; Data for Routine_1
DECL LDAT LCPDATP97={VEL 1.0,ACC 100,APO_DIST 5,APO_FAC 50.0,ORI_TYP #VAR,CIRC_TYP #BASE,JERK_FAC 50.0}
DECL FDAT FP97={TOOL_NO 2,BASE_NO 9,IPO_FRAME #BASE,POINT2[] " ",TQ_STATE FALSE}
DECL E6POS XP97={X 100.000,Y 0.000,Z -100.000,A 0.000,B 0.000,C 0.000}
DECL LDAT LCPDATP98={VEL 0.065,ACC 100,APO_DIST 5,APO_FAC 50.0,ORI_TYP #VAR,CIRC_TYP #BASE,JERK_FAC 50.0}
DECL FDAT FP98={TOOL_NO 2,BASE_NO 9,IPO_FRAME #BASE,POINT2[] " ",TQ_STATE FALSE}
DECL E6POS XP98={X 50.000,Y -2.120,Z -67.490,A 0.000,B 0.000,C -12.000}
DECL LDAT LCPDATP99={VEL 0.065,ACC 100,APO_DIST 5,APO_FAC 50.0,ORI_TYP #VAR,CIRC_TYP #BASE,JERK_FAC 50.0}
DECL FDAT FP99={TOOL_NO 2,BASE_NO 9,IPO_FRAME #BASE,POINT2[] " ",TQ_STATE FALSE}
DECL E6POS XP99={X 0.000,Y -2.120,Z -67.490,A 0.000,B 0.000,C -12.000}
DECL LDAT LCPDATP100={VEL 0.065,ACC 100,APO_DIST 5,APO_FAC 50.0,ORI_TYP #VAR,CIRC_TYP #BASE,JERK_FAC 50.0}
DECL FDAT FP100={TOOL_NO 2,BASE_NO 9,IPO_FRAME #BASE,POINT2[] " ",TQ_STATE FALSE}
DECL E6POS XP100={X -50.000,Y -2.120,Z -67.490,A 0.000,B 0.000,C -12.000}
DECL LDAT LCPDATP101={VEL 0.065,ACC 100,APO_DIST 5,APO_FAC 50.0,ORI_TYP #VAR,CIRC_TYP #BASE,JERK_FAC 50.0}
DECL FDAT FP101={TOOL_NO 2,BASE_NO 9,IPO_FRAME #BASE,POINT2[] " ",TQ_STATE FALSE}
DECL E6POS XP101={X -100.000,Y -2.120,Z -67.490,A 0.000,B 0.000,C -12.000}
DECL LDAT LCPDATP102={VEL 0.088,ACC 100,APO_DIST 5,APO_FAC 50.0,ORI_TYP #VAR,CIRC_TYP #BASE,JERK_FAC 50.0}
DECL FDAT FP102={TOOL_NO 2,BASE_NO 9,IPO_FRAME #BASE,POINT2[] " ",TQ_STATE FALSE}
DECL E6POS XP102={X -100.000,Y 15.760,Z -30.600,A 0.000,B 0.000,C -17.000}
DECL LDAT LCPDATP103={VEL 0.088,ACC 100,APO_DIST 5,APO_FAC 50.0,ORI_TYP #VAR,CIRC_TYP #BASE,JERK_FAC 50.0}
DECL FDAT FP103={TOOL_NO 2,BASE_NO 9,IPO_FRAME #BASE,POINT2[] " ",TQ_STATE FALSE}
DECL E6POS XP103={X -50.000,Y 15.760,Z -30.600,A 0.000,B 0.000,C -17.000}
DECL LDAT LCPDATP104={VEL 0.088,ACC 100,APO_DIST 5,APO_FAC 50.0,ORI_TYP #VAR,CIRC_TYP #BASE,JERK_FAC 50.0}
DECL FDAT FP104={TOOL_NO 2,BASE_NO 9,IPO_FRAME #BASE,POINT2[] " ",TQ_STATE FALSE}
DECL E6POS XP104={X -0.000,Y 15.760,Z -30.600,A 0.000,B 0.000,C -17.000}
DECL LDAT LCPDATP105={VEL 0.088,ACC 100,APO_DIST 5,APO_FAC 50.0,ORI_TYP #VAR,CIRC_TYP #BASE,JERK_FAC 50.0}
DECL FDAT FP105={TOOL_NO 2,BASE_NO 9,IPO_FRAME #BASE,POINT2[] " ",TQ_STATE FALSE}
DECL E6POS XP105={X 50.000,Y 15.760,Z -30.600,A 0.000,B 0.000,C -17.000}
DECL LDAT LCPDATP106={VEL 0.06,ACC 100,APO_DIST 5,APO_FAC 50.0,ORI_TYP #VAR,CIRC_TYP #BASE,JERK_FAC 50.0}
DECL FDAT FP106={TOOL_NO 2,BASE_NO 9,IPO_FRAME #BASE,POINT2[] " ",TQ_STATE FALSE}
DECL E6POS XP106={X 50.000,Y 13.210,Z -73.250,A 0.000,B 0.000,C -22.000}
DECL LDAT LCPDATP107={VEL 0.06,ACC 100,APO_DIST 5,APO_FAC 50.0,ORI_TYP #VAR,CIRC_TYP #BASE,JERK_FAC 50.0}
DECL FDAT FP107={TOOL_NO 2,BASE_NO 9,IPO_FRAME #BASE,POINT2[] " ",TQ_STATE FALSE}
DECL E6POS XP107={X -0.000,Y 13.210,Z -73.250,A 0.000,B 0.000,C -22.000}
DECL LDAT LCPDATP108={VEL 0.06,ACC 100,APO_DIST 5,APO_FAC 50.0,ORI_TYP #VAR,CIRC_TYP #BASE,JERK_FAC 50.0}
DECL FDAT FP108={TOOL_NO 2,BASE_NO 9,IPO_FRAME #BASE,POINT2[] " ",TQ_STATE FALSE}
DECL E6POS XP108={X -50.000,Y 13.210,Z -73.250,A 0.000,B 0.000,C -22.000}
DECL LDAT LCPDATP109={VEL 0.06,ACC 100,APO_DIST 5,APO_FAC 50.0,ORI_TYP #VAR,CIRC_TYP #BASE,JERK_FAC 50.0}
DECL FDAT FP109={TOOL_NO 2,BASE_NO 9,IPO_FRAME #BASE,POINT2[] " ",TQ_STATE FALSE}
DECL E6POS XP109={X -100.000,Y 13.210,Z -73.250,A 0.000,B 0.000,C -22.000}
DECL LDAT LCPDATP110={VEL 0.135,ACC 100,APO_DIST 5,APO_FAC 50.0,ORI_TYP #VAR,CIRC_TYP #BASE,JERK_FAC 50.0}
DECL FDAT FP110={TOOL_NO 2,BASE_NO 9,IPO_FRAME #BASE,POINT2[] " ",TQ_STATE FALSE}
DECL E6POS XP110={X -100.000,Y 40.110,Z -53.550,A 0.000,B 0.000,C -17.000}
DECL LDAT LCPDATP111={VEL 0.135,ACC 100,APO_DIST 5,APO_FAC 50.0,ORI_TYP #VAR,CIRC_TYP #BASE,JERK_FAC 50.0}
DECL FDAT FP111={TOOL_NO 2,BASE_NO 9,IPO_FRAME #BASE,POINT2[] " ",TQ_STATE FALSE}
DECL E6POS XP111={X -50.000,Y 40.110,Z -53.550,A 0.000,B 0.000,C -17.000}
DECL LDAT LCPDATP112={VEL 0.135,ACC 100,APO_DIST 5,APO_FAC 50.0,ORI_TYP #VAR,CIRC_TYP #BASE,JERK_FAC 50.0}
DECL FDAT FP112={TOOL_NO 2,BASE_NO 9,IPO_FRAME #BASE,POINT2[] " ",TQ_STATE FALSE}
DECL E6POS XP112={X -0.000,Y 40.110,Z -53.550,A 0.000,B 0.000,C -17.000}
DECL LDAT LCPDATP113={VEL 0.135,ACC 100,APO_DIST 5,APO_FAC 50.0,ORI_TYP #VAR,CIRC_TYP #BASE,JERK_FAC 50.0}
DECL FDAT FP113={TOOL_NO 2,BASE_NO 9,IPO_FRAME #BASE,POINT2[] " ",TQ_STATE FALSE}
DECL E6POS XP113={X 50.000,Y 40.110,Z -53.550,A 0.000,B 0.000,C -17.000}
DECL LDAT LCPDATP114={VEL 0.119,ACC 100,APO_DIST 5,APO_FAC 50.0,ORI_TYP #VAR,CIRC_TYP #BASE,JERK_FAC 50.0}
DECL FDAT FP114={TOOL_NO 2,BASE_NO 9,IPO_FRAME #BASE,POINT2[] " ",TQ_STATE FALSE}
DECL E6POS XP114={X 50.000,Y 24.230,Z -59.840,A 0.000,B 0.000,C -39.000}
DECL LDAT LCPDATP115={VEL 0.119,ACC 100,APO_DIST 5,APO_FAC 50.0,ORI_TYP #VAR,CIRC_TYP #BASE,JERK_FAC 50.0}
DECL FDAT FP115={TOOL_NO 2,BASE_NO 9,IPO_FRAME #BASE,POINT2[] " ",TQ_STATE FALSE}
DECL E6POS XP115={X -0.000,Y 24.230,Z -59.840,A 0.000,B 0.000,C -39.000}
DECL LDAT LCPDATP116={VEL 0.119,ACC 100,APO_DIST 5,APO_FAC 50.0,ORI_TYP #VAR,CIRC_TYP #BASE,JERK_FAC 50.0}
DECL FDAT FP116={TOOL_NO 2,BASE_NO 9,IPO_FRAME #BASE,POINT2[] " ",TQ_STATE FALSE}
DECL E6POS XP116={X -50.000,Y 24.230,Z -59.840,A 0.000,B 0.000,C -39.000}
DECL LDAT LCPDATP117={VEL 0.119,ACC 100,APO_DIST 5,APO_FAC 50.0,ORI_TYP #VAR,CIRC_TYP #BASE,JERK_FAC 50.0}
DECL FDAT FP117={TOOL_NO 2,BASE_NO 9,IPO_FRAME #BASE,POINT2[] " ",TQ_STATE FALSE}
DECL E6POS XP117={X -100.000,Y 24.230,Z -59.840,A 0.000,B 0.000,C -39.000}
DECL LDAT LCPDATP118={VEL 0.069,ACC 100,APO_DIST 5,APO_FAC 50.0,ORI_TYP #VAR,CIRC_TYP #BASE,JERK_FAC 50.0}
DECL FDAT FP118={TOOL_NO 2,BASE_NO 9,IPO_FRAME #BASE,POINT2[] " ",TQ_STATE FALSE}
DECL E6POS XP118={X -100.000,Y 48.790,Z -52.590,A 0.000,B 0.000,C -36.000}
DECL LDAT LCPDATP119={VEL 0.069,ACC 100,APO_DIST 5,APO_FAC 50.0,ORI_TYP #VAR,CIRC_TYP #BASE,JERK_FAC 50.0}
DECL FDAT FP119={TOOL_NO 2,BASE_NO 9,IPO_FRAME #BASE,POINT2[] " ",TQ_STATE FALSE}
DECL E6POS XP119={X -50.000,Y 48.790,Z -52.590,A 0.000,B 0.000,C -36.000}
DECL LDAT LCPDATP120={VEL 0.069,ACC 100,APO_DIST 5,APO_FAC 50.0,ORI_TYP #VAR,CIRC_TYP #BASE,JERK_FAC 50.0}
DECL FDAT FP120={TOOL_NO 2,BASE_NO 9,IPO_FRAME #BASE,POINT2[] " ",TQ_STATE FALSE}
DECL E6POS XP120={X -0.000,Y 48.790,Z -52.590,A 0.000,B 0.000,C -36.000}
DECL LDAT LCPDATP121={VEL 0.069,ACC 100,APO_DIST 5,APO_FAC 50.0,ORI_TYP #VAR,CIRC_TYP #BASE,JERK_FAC 50.0}
DECL FDAT FP121={TOOL_NO 2,BASE_NO 9,IPO_FRAME #BASE,POINT2[] " ",TQ_STATE FALSE}
DECL E6POS XP121={X 50.000,Y 48.790,Z -52.590,A 0.000,B 0.000,C -36.000}
DECL LDAT LCPDATP122={VEL 0.093,ACC 100,APO_DIST 5,APO_FAC 50.0,ORI_TYP #VAR,CIRC_TYP #BASE,JERK_FAC 50.0}
DECL FDAT FP122={TOOL_NO 2,BASE_NO 9,IPO_FRAME #BASE,POINT2[] " ",TQ_STATE FALSE}
DECL E6POS XP122={X 50.000,Y 91.140,Z -71.110,A 0.000,B 0.000,C -9.000}
DECL LDAT LCPDATP123={VEL 0.093,ACC 100,APO_DIST 5,APO_FAC 50.0,ORI_TYP #VAR,CIRC_TYP #BASE,JERK_FAC 50.0}
DECL FDAT FP123={TOOL_NO 2,BASE_NO 9,IPO_FRAME #BASE,POINT2[] " ",TQ_STATE FALSE}
DECL E6POS XP123={X -0.000,Y 91.140,Z -71.110,A 0.000,B 0.000,C -9.000}
DECL LDAT LCPDATP124={VEL 0.093,ACC 100,APO_DIST 5,APO_FAC 50.0,ORI_TYP #VAR,CIRC_TYP #BASE,JERK_FAC 50.0}
DECL FDAT FP124={TOOL_NO 2,BASE_NO 9,IPO_FRAME #BASE,POINT2[] " ",TQ_STATE FALSE}
DECL E6POS XP124={X -50.000,Y 91.140,Z -71.110,A 0.000,B 0.000,C -9.000}
DECL LDAT LCPDATP125={VEL 0.093,ACC 100,APO_DIST 5,APO_FAC 50.0,ORI_TYP #VAR,CIRC_TYP #BASE,JERK_FAC 50.0}
DECL FDAT FP125={TOOL_NO 2,BASE_NO 9,IPO_FRAME #BASE,POINT2[] " ",TQ_STATE FALSE}
DECL E6POS XP125={X -100.000,Y 91.140,Z -71.110,A 0.000,B 0.000,C -9.000}
DECL LDAT LCPDATP126={VEL 0.072,ACC 100,APO_DIST 5,APO_FAC 50.0,ORI_TYP #VAR,CIRC_TYP #BASE,JERK_FAC 50.0}
DECL FDAT FP126={TOOL_NO 2,BASE_NO 9,IPO_FRAME #BASE,POINT2[] " ",TQ_STATE FALSE}
DECL E6POS XP126={X -100.000,Y 100.110,Z -53.550,A 0.000,B 0.000,C -17.000}
DECL LDAT LCPDATP127={VEL 0.072,ACC 100,APO_DIST 5,APO_FAC 50.0,ORI_TYP #VAR,CIRC_TYP #BASE,JERK_FAC 50.0}
DECL FDAT FP127={TOOL_NO 2,BASE_NO 9,IPO_FRAME #BASE,POINT2[] " ",TQ_STATE FALSE}
DECL E6POS XP127={X -50.000,Y 100.110,Z -53.550,A 0.000,B 0.000,C -17.000}
DECL LDAT LCPDATP128={VEL 0.072,ACC 100,APO_DIST 5,APO_FAC 50.0,ORI_TYP #VAR,CIRC_TYP #BASE,JERK_FAC 50.0}
DECL FDAT FP128={TOOL_NO 2,BASE_NO 9,IPO_FRAME #BASE,POINT2[] " ",TQ_STATE FALSE}
DECL E6POS XP128={X -0.000,Y 100.110,Z -53.550,A 0.000,B 0.000,C -17.000}
DECL LDAT LCPDATP129={VEL 0.072,ACC 100,APO_DIST 5,APO_FAC 50.0,ORI_TYP #VAR,CIRC_TYP #BASE,JERK_FAC 50.0}
DECL FDAT FP129={TOOL_NO 2,BASE_NO 9,IPO_FRAME #BASE,POINT2[] " ",TQ_STATE FALSE}
DECL E6POS XP129={X 50.000,Y 100.110,Z -53.550,A 0.000,B 0.000,C -17.000}
DECL LDAT LCPDATP130={VEL 0.148,ACC 100,APO_DIST 5,APO_FAC 50.0,ORI_TYP #VAR,CIRC_TYP #BASE,JERK_FAC 50.0}
DECL FDAT FP130={TOOL_NO 2,BASE_NO 9,IPO_FRAME #BASE,POINT2[] " ",TQ_STATE FALSE}
DECL E6POS XP130={X 50.000,Y 97.570,Z -52.840,A 0.000,B 0.000,C -33.000}
DECL LDAT LCPDATP131={VEL 0.148,ACC 100,APO_DIST 5,APO_FAC 50.0,ORI_TYP #VAR,CIRC_TYP #BASE,JERK_FAC 50.0}
DECL FDAT FP131={TOOL_NO 2,BASE_NO 9,IPO_FRAME #BASE,POINT2[] " ",TQ_STATE FALSE}
DECL E6POS XP131={X -0.000,Y 97.570,Z -52.840,A 0.000,B 0.000,C -33.000}
DECL LDAT LCPDATP132={VEL 0.148,ACC 100,APO_DIST 5,APO_FAC 50.0,ORI_TYP #VAR,CIRC_TYP #BASE,JERK_FAC 50.0}
DECL FDAT FP132={TOOL_NO 2,BASE_NO 9,IPO_FRAME #BASE,POINT2[] " ",TQ_STATE FALSE}
DECL E6POS XP132={X -50.000,Y 97.570,Z -52.840,A 0.000,B 0.000,C -33.000}
DECL LDAT LCPDATP133={VEL 0.148,ACC 100,APO_DIST 5,APO_FAC 50.0,ORI_TYP #VAR,CIRC_TYP #BASE,JERK_FAC 50.0}
DECL FDAT FP133={TOOL_NO 2,BASE_NO 9,IPO_FRAME #BASE,POINT2[] " ",TQ_STATE FALSE}
DECL E6POS XP133={X -100.000,Y 97.570,Z -52.840,A 0.000,B 0.000,C -33.000}
DECL LDAT LCPDATP134={VEL 0.055,ACC 100,APO_DIST 5,APO_FAC 50.0,ORI_TYP #VAR,CIRC_TYP #BASE,JERK_FAC 50.0}
DECL FDAT FP134={TOOL_NO 2,BASE_NO 9,IPO_FRAME #BASE,POINT2[] " ",TQ_STATE FALSE}
DECL E6POS XP134={X -100.000,Y 134.600,Z -45.600,A 0.000,B 0.000,C -14.000}
DECL LDAT LCPDATP135={VEL 0.055,ACC 100,APO_DIST 5,APO_FAC 50.0,ORI_TYP #VAR,CIRC_TYP #BASE,JERK_FAC 50.0}
DECL FDAT FP135={TOOL_NO 2,BASE_NO 9,IPO_FRAME #BASE,POINT2[] " ",TQ_STATE FALSE}
DECL E6POS XP135={X -50.000,Y 134.600,Z -45.600,A 0.000,B 0.000,C -14.000}
DECL LDAT LCPDATP136={VEL 0.055,ACC 100,APO_DIST 5,APO_FAC 50.0,ORI_TYP #VAR,CIRC_TYP #BASE,JERK_FAC 50.0}
DECL FDAT FP136={TOOL_NO 2,BASE_NO 9,IPO_FRAME #BASE,POINT2[] " ",TQ_STATE FALSE}
DECL E6POS XP136={X -0.000,Y 134.600,Z -45.600,A 0.000,B 0.000,C -14.000}
DECL LDAT LCPDATP137={VEL 0.055,ACC 100,APO_DIST 5,APO_FAC 50.0,ORI_TYP #VAR,CIRC_TYP #BASE,JERK_FAC 50.0}
DECL FDAT FP137={TOOL_NO 2,BASE_NO 9,IPO_FRAME #BASE,POINT2[] " ",TQ_STATE FALSE}
DECL E6POS XP137={X 50.000,Y 134.600,Z -45.600,A 0.000,B 0.000,C -14.000}
DECL LDAT LCPDATP138={VEL 0.149,ACC 100,APO_DIST 5,APO_FAC 50.0,ORI_TYP #VAR,CIRC_TYP #BASE,JERK_FAC 50.0}
DECL FDAT FP138={TOOL_NO 2,BASE_NO 9,IPO_FRAME #BASE,POINT2[] " ",TQ_STATE FALSE}
DECL E6POS XP138={X 50.000,Y 142.850,Z -89.640,A 0.000,B 0.000,C -13.000}
DECL LDAT LCPDATP139={VEL 0.149,ACC 100,APO_DIST 5,APO_FAC 50.0,ORI_TYP #VAR,CIRC_TYP #BASE,JERK_FAC 50.0}
DECL FDAT FP139={TOOL_NO 2,BASE_NO 9,IPO_FRAME #BASE,POINT2[] " ",TQ_STATE FALSE}
DECL E6POS XP139={X -0.000,Y 142.850,Z -89.640,A 0.000,B 0.000,C -13.000}
DECL LDAT LCPDATP140={VEL 0.149,ACC 100,APO_DIST 5,APO_FAC 50.0,ORI_TYP #VAR,CIRC_TYP #BASE,JERK_FAC 50.0}
DECL FDAT FP140={TOOL_NO 2,BASE_NO 9,IPO_FRAME #BASE,POINT2[] " ",TQ_STATE FALSE}
DECL E6POS XP140={X -50.000,Y 142.850,Z -89.640,A 0.000,B 0.000,C -13.000}
DECL LDAT LCPDATP141={VEL 0.149,ACC 100,APO_DIST 5,APO_FAC 50.0,ORI_TYP #VAR,CIRC_TYP #BASE,JERK_FAC 50.0}
DECL FDAT FP141={TOOL_NO 2,BASE_NO 9,IPO_FRAME #BASE,POINT2[] " ",TQ_STATE FALSE}
DECL E6POS XP141={X -100.000,Y 142.850,Z -89.640,A 0.000,B 0.000,C -13.000}
DECL LDAT LCPDATP142={VEL 0.101,ACC 100,APO_DIST 5,APO_FAC 50.0,ORI_TYP #VAR,CIRC_TYP #BASE,JERK_FAC 50.0}
DECL FDAT FP142={TOOL_NO 2,BASE_NO 9,IPO_FRAME #BASE,POINT2[] " ",TQ_STATE FALSE}
DECL E6POS XP142={X -100.000,Y 141.950,Z -67.100,A 0.000,B 0.000,C -28.000}
DECL LDAT LCPDATP143={VEL 0.101,ACC 100,APO_DIST 5,APO_FAC 50.0,ORI_TYP #VAR,CIRC_TYP #BASE,JERK_FAC 50.0}
DECL FDAT FP143={TOOL_NO 2,BASE_NO 9,IPO_FRAME #BASE,POINT2[] " ",TQ_STATE FALSE}
DECL E6POS XP143={X -50.000,Y 141.950,Z -67.100,A 0.000,B 0.000,C -28.000}
DECL LDAT LCPDATP144={VEL 0.101,ACC 100,APO_DIST 5,APO_FAC 50.0,ORI_TYP #VAR,CIRC_TYP #BASE,JERK_FAC 50.0}
DECL FDAT FP144={TOOL_NO 2,BASE_NO 9,IPO_FRAME #BASE,POINT2[] " ",TQ_STATE FALSE}
DECL E6POS XP144={X -0.000,Y 141.950,Z -67.100,A 0.000,B 0.000,C -28.000}
DECL LDAT LCPDATP145={VEL 0.101,ACC 100,APO_DIST 5,APO_FAC 50.0,ORI_TYP #VAR,CIRC_TYP #BASE,JERK_FAC 50.0}
DECL FDAT FP145={TOOL_NO 2,BASE_NO 9,IPO_FRAME #BASE,POINT2[] " ",TQ_STATE FALSE}
DECL E6POS XP145={X 50.000,Y 141.950,Z -67.100,A 0.000,B 0.000,C -28.000}
DECL LDAT LCPDATP146={VEL 0.071,ACC 100,APO_DIST 5,APO_FAC 50.0,ORI_TYP #VAR,CIRC_TYP #BASE,JERK_FAC 50.0}
DECL FDAT FP146={TOOL_NO 2,BASE_NO 9,IPO_FRAME #BASE,POINT2[] " ",TQ_STATE FALSE}
DECL E6POS XP146={X 50.000,Y 189.020,Z -32.980,A 0.000,B 0.000,C -2.000}
DECL LDAT LCPDATP147={VEL 0.071,ACC 100,APO_DIST 5,APO_FAC 50.0,ORI_TYP #VAR,CIRC_TYP #BASE,JERK_FAC 50.0}
DECL FDAT FP147={TOOL_NO 2,BASE_NO 9,IPO_FRAME #BASE,POINT2[] " ",TQ_STATE FALSE}
DECL E6POS XP147={X -0.000,Y 189.020,Z -32.980,A 0.000,B 0.000,C -2.000}
DECL LDAT LCPDATP148={VEL 0.071,ACC 100,APO_DIST 5,APO_FAC 50.0,ORI_TYP #VAR,CIRC_TYP #BASE,JERK_FAC 50.0}
DECL FDAT FP148={TOOL_NO 2,BASE_NO 9,IPO_FRAME #BASE,POINT2[] " ",TQ_STATE FALSE}
DECL E6POS XP148={X -50.000,Y 189.020,Z -32.980,A 0.000,B 0.000,C -2.000}
DECL LDAT LCPDATP149={VEL 0.071,ACC 100,APO_DIST 5,APO_FAC 50.0,ORI_TYP #VAR,CIRC_TYP #BASE,JERK_FAC 50.0}
DECL FDAT FP149={TOOL_NO 2,BASE_NO 9,IPO_FRAME #BASE,POINT2[] " ",TQ_STATE FALSE}
DECL E6POS XP149={X -100.000,Y 189.020,Z -32.980,A 0.000,B 0.000,C -2.000}
DECL LDAT LCPDATP150={VEL 0.121,ACC 100,APO_DIST 5,APO_FAC 50.0,ORI_TYP #VAR,CIRC_TYP #BASE,JERK_FAC 50.0}
DECL FDAT FP150={TOOL_NO 2,BASE_NO 9,IPO_FRAME #BASE,POINT2[] " ",TQ_STATE FALSE}
DECL E6POS XP150={X -100.000,Y 199.670,Z -30.530,A 0.000,B 0.000,C -10.000}
DECL LDAT LCPDATP151={VEL 0.121,ACC 100,APO_DIST 5,APO_FAC 50.0,ORI_TYP #VAR,CIRC_TYP #BASE,JERK_FAC 50.0}
DECL FDAT FP151={TOOL_NO 2,BASE_NO 9,IPO_FRAME #BASE,POINT2[] " ",TQ_STATE FALSE}
DECL E6POS XP151={X -50.000,Y 199.670,Z -30.530,A 0.000,B 0.000,C -10.000}
DECL LDAT LCPDATP152={VEL 0.121,ACC 100,APO_DIST 5,APO_FAC 50.0,ORI_TYP #VAR,CIRC_TYP #BASE,JERK_FAC 50.0}
DECL FDAT FP152={TOOL_NO 2,BASE_NO 9,IPO_FRAME #BASE,POINT2[] " ",TQ_STATE FALSE}
DECL E6POS XP152={X -0.000,Y 199.670,Z -30.530,A 0.000,B 0.000,C -10.000}
DECL LDAT LCPDATP153={VEL 0.121,ACC 100,APO_DIST 5,APO_FAC 50.0,ORI_TYP #VAR,CIRC_TYP #BASE,JERK_FAC 50.0}
DECL FDAT FP153={TOOL_NO 2,BASE_NO 9,IPO_FRAME #BASE,POINT2[] " ",TQ_STATE FALSE}
DECL E6POS XP153={X 50.000,Y 199.670,Z -30.530,A 0.000,B 0.000,C -10.000}
DECL LDAT LCPDATP154={VEL 0.061,ACC 100,APO_DIST 5,APO_FAC 50.0,ORI_TYP #VAR,CIRC_TYP #BASE,JERK_FAC 50.0}
DECL FDAT FP154={TOOL_NO 2,BASE_NO 9,IPO_FRAME #BASE,POINT2[] " ",TQ_STATE FALSE}
DECL E6POS XP154={X 50.000,Y 202.790,Z -30.310,A 0.000,B 0.000,C -30.000}
DECL LDAT LCPDATP155={VEL 0.061,ACC 100,APO_DIST 5,APO_FAC 50.0,ORI_TYP #VAR,CIRC_TYP #BASE,JERK_FAC 50.0}
DECL FDAT FP155={TOOL_NO 2,BASE_NO 9,IPO_FRAME #BASE,POINT2[] " ",TQ_STATE FALSE}
DECL E6POS XP155={X -0.000,Y 202.790,Z -30.310,A 0.000,B 0.000,C -30.000}
DECL LDAT LCPDATP156={VEL 0.061,ACC 100,APO_DIST 5,APO_FAC 50.0,ORI_TYP #VAR,CIRC_TYP #BASE,JERK_FAC 50.0}
DECL FDAT FP156={TOOL_NO 2,BASE_NO 9,IPO_FRAME #BASE,POINT2[] " ",TQ_STATE FALSE}
DECL E6POS XP156={X -50.000,Y 202.790,Z -30.310,A 0.000,B 0.000,C -30.000}
DECL LDAT LCPDATP157={VEL 0.061,ACC 100,APO_DIST 5,APO_FAC 50.0,ORI_TYP #VAR,CIRC_TYP #BASE,JERK_FAC 50.0}
DECL FDAT FP157={TOOL_NO 2,BASE_NO 9,IPO_FRAME #BASE,POINT2[] " ",TQ_STATE FALSE}
DECL E6POS XP157={X -100.000,Y 202.790,Z -30.310,A 0.000,B 0.000,C -30.000}
DECL LDAT LCPDATP158={VEL 0.5,ACC 100,APO_DIST 5,APO_FAC 50.0,ORI_TYP #VAR,CIRC_TYP #BASE,JERK_FAC 50.0}
DECL FDAT FP158={TOOL_NO 2,BASE_NO 9,IPO_FRAME #BASE,POINT2[] " ",TQ_STATE FALSE}
DECL E6POS XP158={X -150.000,Y 220.290,Z -50.000,A 0.000,B 0.000,C 0.000}
DECL LDAT LCPDATP159={VEL 1.0,ACC 100,APO_DIST 5,APO_FAC 50.0,ORI_TYP #VAR,CIRC_TYP #BASE,JERK_FAC 50.0}
DECL FDAT FP159={TOOL_NO 2,BASE_NO 9,IPO_FRAME #BASE,POINT2[] " ",TQ_STATE FALSE}
DECL E6POS XP159={X -150.000,Y 260.000,Z -20.000,A 0.000,B 0.000,C 0.000}
DECL LDAT LCPDATP160={VEL 1.0,ACC 100,APO_DIST 5,APO_FAC 50.0,ORI_TYP #VAR,CIRC_TYP #BASE,JERK_FAC 50.0}
DECL FDAT FP160={TOOL_NO 2,BASE_NO 9,IPO_FRAME #BASE,POINT2[] " ",TQ_STATE FALSE}
DECL E6POS XP160={X 100.000,Y 260.000,Z -20.000,A 0.000,B 0.000,C 0.000}
;ENDDAT for Routine_1


; Data for Routine_2
DECL LDAT LCPDATP161={VEL 1.0,ACC 100,APO_DIST 5,APO_FAC 50.0,ORI_TYP #VAR,CIRC_TYP #BASE,JERK_FAC 50.0}
DECL FDAT FP161={TOOL_NO 2,BASE_NO 8,IPO_FRAME #BASE,POINT2[] " ",TQ_STATE FALSE}
DECL E6POS XP161={X 100.000,Y 0.000,Z -100.000,A 0.000,B 0.000,C 0.000}
DECL LDAT LCPDATP162={VEL 0.123,ACC 100,APO_DIST 5,APO_FAC 50.0,ORI_TYP #VAR,CIRC_TYP #BASE,JERK_FAC 50.0}
DECL FDAT FP162={TOOL_NO 2,BASE_NO 8,IPO_FRAME #BASE,POINT2[] " ",TQ_STATE FALSE}
DECL E6POS XP162={X 50.000,Y -12.510,Z -68.600,A 0.000,B 0.000,C -20.000}
DECL LDAT LCPDATP163={VEL 0.123,ACC 100,APO_DIST 5,APO_FAC 50.0,ORI_TYP #VAR,CIRC_TYP #BASE,JERK_FAC 50.0}
DECL FDAT FP163={TOOL_NO 2,BASE_NO 8,IPO_FRAME #BASE,POINT2[] " ",TQ_STATE FALSE}
DECL E6POS XP163={X 0.000,Y -12.510,Z -68.600,A 0.000,B 0.000,C -20.000}
DECL LDAT LCPDATP164={VEL 0.123,ACC 100,APO_DIST 5,APO_FAC 50.0,ORI_TYP #VAR,CIRC_TYP #BASE,JERK_FAC 50.0}
DECL FDAT FP164={TOOL_NO 2,BASE_NO 8,IPO_FRAME #BASE,POINT2[] " ",TQ_STATE FALSE}
DECL E6POS XP164={X -50.000,Y -12.510,Z -68.600,A 0.000,B 0.000,C -20.000}
DECL LDAT LCPDATP165={VEL 0.123,ACC 100,APO_DIST 5,APO_FAC 50.0,ORI_TYP #VAR,CIRC_TYP #BASE,JERK_FAC 50.0}
DECL FDAT FP165={TOOL_NO 2,BASE_NO 8,IPO_FRAME #BASE,POINT2[] " ",TQ_STATE FALSE}
DECL E6POS XP165={X -100.000,Y -12.510,Z -68.600,A 0.000,B 0.000,C -20.000}
DECL LDAT LCPDATP166={VEL 0.128,ACC 100,APO_DIST 5,APO_FAC 50.0,ORI_TYP #VAR,CIRC_TYP #BASE,JERK_FAC 50.0}
DECL FDAT FP166={TOOL_NO 2,BASE_NO 8,IPO_FRAME #BASE,POINT2[] " ",TQ_STATE FALSE}
DECL E6POS XP166={X -100.000,Y -8.150,Z -77.940,A 0.000,B 0.000,C -25.000}
DECL LDAT LCPDATP167={VEL 0.128,ACC 100,APO_DIST 5,APO_FAC 50.0,ORI_TYP #VAR,CIRC_TYP #BASE,JERK_FAC 50.0}
DECL FDAT FP167={TOOL_NO 2,BASE_NO 8,IPO_FRAME #BASE,POINT2[] " ",TQ_STATE FALSE}
DECL E6POS XP167={X -50.000,Y -8.150,Z -77.940,A 0.000,B 0.000,C -25.000}
DECL LDAT LCPDATP168={VEL 0.128,ACC 100,APO_DIST 5,APO_FAC 50.0,ORI_TYP #VAR,CIRC_TYP #BASE,JERK_FAC 50.0}
DECL FDAT FP168={TOOL_NO 2,BASE_NO 8,IPO_FRAME #BASE,POINT2[] " ",TQ_STATE FALSE}
DECL E6POS XP168={X 0.000,Y -8.150,Z -77.940,A 0.000,B 0.000,C -25.000}
DECL LDAT LCPDATP169={VEL 0.128,ACC 100,APO_DIST 5,APO_FAC 50.0,ORI_TYP #VAR,CIRC_TYP #BASE,JERK_FAC 50.0}
DECL FDAT FP169={TOOL_NO 2,BASE_NO 8,IPO_FRAME #BASE,POINT2[] " ",TQ_STATE FALSE}
DECL E6POS XP169={X 50.000,Y -8.150,Z -77.940,A 0.000,B 0.000,C -25.000}
DECL LDAT LCPDATP170={VEL 0.103,ACC 100,APO_DIST 5,APO_FAC 50.0,ORI_TYP #VAR,CIRC_TYP #BASE,JERK_FAC 50.0}
DECL FDAT FP170={TOOL_NO 2,BASE_NO 8,IPO_FRAME #BASE,POINT2[] " ",TQ_STATE FALSE}
DECL E6POS XP170={X 50.000,Y 41.710,Z -60.000,A 0.000,B 0.000,C 0.000}
DECL LDAT LCPDATP171={VEL 0.103,ACC 100,APO_DIST 5,APO_FAC 50.0,ORI_TYP #VAR,CIRC_TYP #BASE,JERK_FAC 50.0}
DECL FDAT FP171={TOOL_NO 2,BASE_NO 8,IPO_FRAME #BASE,POINT2[] " ",TQ_STATE FALSE}
DECL E6POS XP171={X -0.000,Y 41.710,Z -60.000,A 0.000,B 0.000,C 0.000}
DECL LDAT LCPDATP172={VEL 0.103,ACC 100,APO_DIST 5,APO_FAC 50.0,ORI_TYP #VAR,CIRC_TYP #BASE,JERK_FAC 50.0}
DECL FDAT FP172={TOOL_NO 2,BASE_NO 8,IPO_FRAME #BASE,POINT2[] " ",TQ_STATE FALSE}
DECL E6POS XP172={X -50.000,Y 41.710,Z -60.000,A 0.000,B 0.000,C 0.000}
DECL LDAT LCPDATP173={VEL 0.103,ACC 100,APO_DIST 5,APO_FAC 50.0,ORI_TYP #VAR,CIRC_TYP #BASE,JERK_FAC 50.0}
DECL FDAT FP173={TOOL_NO 2,BASE_NO 8,IPO_FRAME #BASE,POINT2[] " ",TQ_STATE FALSE}
DECL E6POS XP173={X -100.000,Y 41.710,Z -60.000,A 0.000,B 0.000,C 0.000}
DECL LDAT LCPDATP174={VEL 0.108,ACC 100,APO_DIST 5,APO_FAC 50.0,ORI_TYP #VAR,CIRC_TYP #BASE,JERK_FAC 50.0}
DECL FDAT FP174={TOOL_NO 2,BASE_NO 8,IPO_FRAME #BASE,POINT2[] " ",TQ_STATE FALSE}
DECL E6POS XP174={X -100.000,Y 43.810,Z -45.400,A 0.000,B 0.000,C -15.000}
DECL LDAT LCPDATP175={VEL 0.108,ACC 100,APO_DIST 5,APO_FAC 50.0,ORI_TYP #VAR,CIRC_TYP #BASE,JERK_FAC 50.0}
DECL FDAT FP175={TOOL_NO 2,BASE_NO 8,IPO_FRAME #BASE,POINT2[] " ",TQ_STATE FALSE}
DECL E6POS XP175={X -50.000,Y 43.810,Z -45.400,A 0.000,B 0.000,C -15.000}
DECL LDAT LCPDATP176={VEL 0.108,ACC 100,APO_DIST 5,APO_FAC 50.0,ORI_TYP #VAR,CIRC_TYP #BASE,JERK_FAC 50.0}
DECL FDAT FP176={TOOL_NO 2,BASE_NO 8,IPO_FRAME #BASE,POINT2[] " ",TQ_STATE FALSE}
DECL E6POS XP176={X -0.000,Y 43.810,Z -45.400,A 0.000,B 0.000,C -15.000}
DECL LDAT LCPDATP177={VEL 0.108,ACC 100,APO_DIST 5,APO_FAC 50.0,ORI_TYP #VAR,CIRC_TYP #BASE,JERK_FAC 50.0}
DECL FDAT FP177={TOOL_NO 2,BASE_NO 8,IPO_FRAME #BASE,POINT2[] " ",TQ_STATE FALSE}
DECL E6POS XP177={X 50.000,Y 43.810,Z -45.400,A 0.000,B 0.000,C -15.000}
DECL LDAT LCPDATP178={VEL 0.095,ACC 100,APO_DIST 5,APO_FAC 50.0,ORI_TYP #VAR,CIRC_TYP #BASE,JERK_FAC 50.0}
DECL FDAT FP178={TOOL_NO 2,BASE_NO 8,IPO_FRAME #BASE,POINT2[] " ",TQ_STATE FALSE}
DECL E6POS XP178={X 50.000,Y 50.270,Z -49.710,A 0.000,B 0.000,C -23.000}
DECL LDAT LCPDATP179={VEL 0.095,ACC 100,APO_DIST 5,APO_FAC 50.0,ORI_TYP #VAR,CIRC_TYP #BASE,JERK_FAC 50.0}
DECL FDAT FP179={TOOL_NO 2,BASE_NO 8,IPO_FRAME #BASE,POINT2[] " ",TQ_STATE FALSE}
DECL E6POS XP179={X -0.000,Y 50.270,Z -49.710,A 0.000,B 0.000,C -23.000}
DECL LDAT LCPDATP180={VEL 0.095,ACC 100,APO_DIST 5,APO_FAC 50.0,ORI_TYP #VAR,CIRC_TYP #BASE,JERK_FAC 50.0}
DECL FDAT FP180={TOOL_NO 2,BASE_NO 8,IPO_FRAME #BASE,POINT2[] " ",TQ_STATE FALSE}
DECL E6POS XP180={X -50.000,Y 50.270,Z -49.710,A 0.000,B 0.000,C -23.000}
DECL LDAT LCPDATP181={VEL 0.095,ACC 100,APO_DIST 5,APO_FAC 50.0,ORI_TYP #VAR,CIRC_TYP #BASE,JERK_FAC 50.0}
DECL FDAT FP181={TOOL_NO 2,BASE_NO 8,IPO_FRAME #BASE,POINT2[] " ",TQ_STATE FALSE}
DECL E6POS XP181={X -100.000,Y 50.270,Z -49.710,A 0.000,B 0.000,C -23.000}
DECL LDAT LCPDATP182={VEL 0.142,ACC 100,APO_DIST 5,APO_FAC 50.0,ORI_TYP #VAR,CIRC_TYP #BASE,JERK_FAC 50.0}
DECL FDAT FP182={TOOL_NO 2,BASE_NO 8,IPO_FRAME #BASE,POINT2[] " ",TQ_STATE FALSE}
DECL E6POS XP182={X -100.000,Y 77.240,Z -35.080,A 0.000,B 0.000,C -13.000}
DECL LDAT LCPDATP183={VEL 0.142,ACC 100,APO_DIST 5,APO_FAC 50.0,ORI_TYP #VAR,CIRC_TYP #BASE,JERK_FAC 50.0}
DECL FDAT FP183={TOOL_NO 2,BASE_NO 8,IPO_FRAME #BASE,POINT2[] " ",TQ_STATE FALSE}
DECL E6POS XP183={X -50.000,Y 77.240,Z -35.080,A 0.000,B 0.000,C -13.000}
DECL LDAT LCPDATP184={VEL 0.142,ACC 100,APO_DIST 5,APO_FAC 50.0,ORI_TYP #VAR,CIRC_TYP #BASE,JERK_FAC 50.0}
DECL FDAT FP184={TOOL_NO 2,BASE_NO 8,IPO_FRAME #BASE,POINT2[] " ",TQ_STATE FALSE}
DECL E6POS XP184={X -0.000,Y 77.240,Z -35.080,A 0.000,B 0.000,C -13.000}
DECL LDAT LCPDATP185={VEL 0.142,ACC 100,APO_DIST 5,APO_FAC 50.0,ORI_TYP #VAR,CIRC_TYP #BASE,JERK_FAC 50.0}
DECL FDAT FP185={TOOL_NO 2,BASE_NO 8,IPO_FRAME #BASE,POINT2[] " ",TQ_STATE FALSE}
DECL E6POS XP185={X 50.000,Y 77.240,Z -35.080,A 0.000,B 0.000,C -13.000}
DECL LDAT LCPDATP186={VEL 0.142,ACC 100,APO_DIST 5,APO_FAC 50.0,ORI_TYP #VAR,CIRC_TYP #BASE,JERK_FAC 50.0}
DECL FDAT FP186={TOOL_NO 2,BASE_NO 8,IPO_FRAME #BASE,POINT2[] " ",TQ_STATE FALSE}
DECL E6POS XP186={X 50.000,Y 94.780,Z -73.590,A 0.000,B 0.000,C -6.000}
DECL LDAT LCPDATP187={VEL 0.142,ACC 100,APO_DIST 5,APO_FAC 50.0,ORI_TYP #VAR,CIRC_TYP #BASE,JERK_FAC 50.0}
DECL FDAT FP187={TOOL_NO 2,BASE_NO 8,IPO_FRAME #BASE,POINT2[] " ",TQ_STATE FALSE}
DECL E6POS XP187={X -0.000,Y 94.780,Z -73.590,A 0.000,B 0.000,C -6.000}
DECL LDAT LCPDATP188={VEL 0.142,ACC 100,APO_DIST 5,APO_FAC 50.0,ORI_TYP #VAR,CIRC_TYP #BASE,JERK_FAC 50.0}
DECL FDAT FP188={TOOL_NO 2,BASE_NO 8,IPO_FRAME #BASE,POINT2[] " ",TQ_STATE FALSE}
DECL E6POS XP188={X -50.000,Y 94.780,Z -73.590,A 0.000,B 0.000,C -6.000}
DECL LDAT LCPDATP189={VEL 0.142,ACC 100,APO_DIST 5,APO_FAC 50.0,ORI_TYP #VAR,CIRC_TYP #BASE,JERK_FAC 50.0}
DECL FDAT FP189={TOOL_NO 2,BASE_NO 8,IPO_FRAME #BASE,POINT2[] " ",TQ_STATE FALSE}
DECL E6POS XP189={X -100.000,Y 94.780,Z -73.590,A 0.000,B 0.000,C -6.000}
DECL LDAT LCPDATP190={VEL 0.064,ACC 100,APO_DIST 5,APO_FAC 50.0,ORI_TYP #VAR,CIRC_TYP #BASE,JERK_FAC 50.0}
DECL FDAT FP190={TOOL_NO 2,BASE_NO 8,IPO_FRAME #BASE,POINT2[] " ",TQ_STATE FALSE}
DECL E6POS XP190={X -100.000,Y 84.800,Z -40.190,A 0.000,B 0.000,C -38.000}
DECL LDAT LCPDATP191={VEL 0.064,ACC 100,APO_DIST 5,APO_FAC 50.0,ORI_TYP #VAR,CIRC_TYP #BASE,JERK_FAC 50.0}
DECL FDAT FP191={TOOL_NO 2,BASE_NO 8,IPO_FRAME #BASE,POINT2[] " ",TQ_STATE FALSE}
DECL E6POS XP191={X -50.000,Y 84.800,Z -40.190,A 0.000,B 0.000,C -38.000}
DECL LDAT LCPDATP192={VEL 0.064,ACC 100,APO_DIST 5,APO_FAC 50.0,ORI_TYP #VAR,CIRC_TYP #BASE,JERK_FAC 50.0}
DECL FDAT FP192={TOOL_NO 2,BASE_NO 8,IPO_FRAME #BASE,POINT2[] " ",TQ_STATE FALSE}
DECL E6POS XP192={X -0.000,Y 84.800,Z -40.190,A 0.000,B 0.000,C -38.000}
DECL LDAT LCPDATP193={VEL 0.064,ACC 100,APO_DIST 5,APO_FAC 50.0,ORI_TYP #VAR,CIRC_TYP #BASE,JERK_FAC 50.0}
DECL FDAT FP193={TOOL_NO 2,BASE_NO 8,IPO_FRAME #BASE,POINT2[] " ",TQ_STATE FALSE}
DECL E6POS XP193={X 50.000,Y 84.800,Z -40.190,A 0.000,B 0.000,C -38.000}
DECL LDAT LCPDATP194={VEL 0.055,ACC 100,APO_DIST 5,APO_FAC 50.0,ORI_TYP #VAR,CIRC_TYP #BASE,JERK_FAC 50.0}
DECL FDAT FP194={TOOL_NO 2,BASE_NO 8,IPO_FRAME #BASE,POINT2[] " ",TQ_STATE FALSE}
DECL E6POS XP194={X 50.000,Y 76.790,Z -69.940,A 0.000,B 0.000,C -39.000}
DECL LDAT LCPDATP195={VEL 0.055,ACC 100,APO_DIST 5,APO_FAC 50.0,ORI_TYP #VAR,CIRC_TYP #BASE,JERK_FAC 50.0}
DECL FDAT FP195={TOOL_NO 2,BASE_NO 8,IPO_FRAME #BASE,POINT2[] " ",TQ_STATE FALSE}
DECL E6POS XP195={X -0.000,Y 76.790,Z -69.940,A 0.000,B 0.000,C -39.000}
DECL LDAT LCPDATP196={VEL 0.055,ACC 100,APO_DIST 5,APO_FAC 50.0,ORI_TYP #VAR,CIRC_TYP #BASE,JERK_FAC 50.0}
DECL FDAT FP196={TOOL_NO 2,BASE_NO 8,IPO_FRAME #BASE,POINT2[] " ",TQ_STATE FALSE}
DECL E6POS XP196={X -50.000,Y 76.790,Z -69.940,A 0.000,B 0.000,C -39.000}
DECL LDAT LCPDATP197={VEL 0.055,ACC 100,APO_DIST 5,APO_FAC 50.0,ORI_TYP #VAR,CIRC_TYP #BASE,JERK_FAC 50.0}
DECL FDAT FP197={TOOL_NO 2,BASE_NO 8,IPO_FRAME #BASE,POINT2[] " ",TQ_STATE FALSE}
DECL E6POS XP197={X -100.000,Y 76.790,Z -69.940,A 0.000,B 0.000,C -39.000}
DECL LDAT LCPDATP198={VEL 0.12,ACC 100,APO_DIST 5,APO_FAC 50.0,ORI_TYP #VAR,CIRC_TYP #BASE,JERK_FAC 50.0}
DECL FDAT FP198={TOOL_NO 2,BASE_NO 8,IPO_FRAME #BASE,POINT2[] " ",TQ_STATE FALSE}
DECL E6POS XP198={X -100.000,Y 132.190,Z -81.480,A 0.000,B 0.000,C -11.000}
DECL LDAT LCPDATP199={VEL 0.12,ACC 100,APO_DIST 5,APO_FAC 50.0,ORI_TYP #VAR,CIRC_TYP #BASE,JERK_FAC 50.0}
DECL FDAT FP199={TOOL_NO 2,BASE_NO 8,IPO_FRAME #BASE,POINT2[] " ",TQ_STATE FALSE}
DECL E6POS XP199={X -50.000,Y 132.190,Z -81.480,A 0.000,B 0.000,C -11.000}
DECL LDAT LCPDATP200={VEL 0.12,ACC 100,APO_DIST 5,APO_FAC 50.0,ORI_TYP #VAR,CIRC_TYP #BASE,JERK_FAC 50.0}
DECL FDAT FP200={TOOL_NO 2,BASE_NO 8,IPO_FRAME #BASE,POINT2[] " ",TQ_STATE FALSE}
DECL E6POS XP200={X -0.000,Y 132.190,Z -81.480,A 0.000,B 0.000,C -11.000}
DECL LDAT LCPDATP201={VEL 0.12,ACC 100,APO_DIST 5,APO_FAC 50.0,ORI_TYP #VAR,CIRC_TYP #BASE,JERK_FAC 50.0}
DECL FDAT FP201={TOOL_NO 2,BASE_NO 8,IPO_FRAME #BASE,POINT2[] " ",TQ_STATE FALSE}
DECL E6POS XP201={X 50.000,Y 132.190,Z -81.480,A 0.000,B 0.000,C -11.000}
DECL LDAT LCPDATP202={VEL 0.081,ACC 100,APO_DIST 5,APO_FAC 50.0,ORI_TYP #VAR,CIRC_TYP #BASE,JERK_FAC 50.0}
DECL FDAT FP202={TOOL_NO 2,BASE_NO 8,IPO_FRAME #BASE,POINT2[] " ",TQ_STATE FALSE}
DECL E6POS XP202={X 50.000,Y 124.070,Z -69.970,A 0.000,B 0.000,C -29.000}
DECL LDAT LCPDATP203={VEL 0.081,ACC 100,APO_DIST 5,APO_FAC 50.0,ORI_TYP #VAR,CIRC_TYP #BASE,JERK_FAC 50.0}
DECL FDAT FP203={TOOL_NO 2,BASE_NO 8,IPO_FRAME #BASE,POINT2[] " ",TQ_STATE FALSE}
DECL E6POS XP203={X -0.000,Y 124.070,Z -69.970,A 0.000,B 0.000,C -29.000}
DECL LDAT LCPDATP204={VEL 0.081,ACC 100,APO_DIST 5,APO_FAC 50.0,ORI_TYP #VAR,CIRC_TYP #BASE,JERK_FAC 50.0}
DECL FDAT FP204={TOOL_NO 2,BASE_NO 8,IPO_FRAME #BASE,POINT2[] " ",TQ_STATE FALSE}
DECL E6POS XP204={X -50.000,Y 124.070,Z -69.970,A 0.000,B 0.000,C -29.000}
DECL LDAT LCPDATP205={VEL 0.081,ACC 100,APO_DIST 5,APO_FAC 50.0,ORI_TYP #VAR,CIRC_TYP #BASE,JERK_FAC 50.0}
DECL FDAT FP205={TOOL_NO 2,BASE_NO 8,IPO_FRAME #BASE,POINT2[] " ",TQ_STATE FALSE}
DECL E6POS XP205={X -100.000,Y 124.070,Z -69.970,A 0.000,B 0.000,C -29.000}
DECL LDAT LCPDATP206={VEL 0.147,ACC 100,APO_DIST 5,APO_FAC 50.0,ORI_TYP #VAR,CIRC_TYP #BASE,JERK_FAC 50.0}
DECL FDAT FP206={TOOL_NO 2,BASE_NO 8,IPO_FRAME #BASE,POINT2[] " ",TQ_STATE FALSE}
DECL E6POS XP206={X -100.000,Y 170.770,Z -52.710,A 0.000,B 0.000,C -6.000}
DECL LDAT LCPDATP207={VEL 0.147,ACC 100,APO_DIST 5,APO_FAC 50.0,ORI_TYP #VAR,CIRC_TYP #BASE,JERK_FAC 50.0}
DECL FDAT FP207={TOOL_NO 2,BASE_NO 8,IPO_FRAME #BASE,POINT2[] " ",TQ_STATE FALSE}
DECL E6POS XP207={X -50.000,Y 170.770,Z -52.710,A 0.000,B 0.000,C -6.000}
DECL LDAT LCPDATP208={VEL 0.147,ACC 100,APO_DIST 5,APO_FAC 50.0,ORI_TYP #VAR,CIRC_TYP #BASE,JERK_FAC 50.0}
DECL FDAT FP208={TOOL_NO 2,BASE_NO 8,IPO_FRAME #BASE,POINT2[] " ",TQ_STATE FALSE}
DECL E6POS XP208={X -0.000,Y 170.770,Z -52.710,A 0.000,B 0.000,C -6.000}
DECL LDAT LCPDATP209={VEL 0.147,ACC 100,APO_DIST 5,APO_FAC 50.0,ORI_TYP #VAR,CIRC_TYP #BASE,JERK_FAC 50.0}
DECL FDAT FP209={TOOL_NO 2,BASE_NO 8,IPO_FRAME #BASE,POINT2[] " ",TQ_STATE FALSE}
DECL E6POS XP209={X 50.000,Y 170.770,Z -52.710,A 0.000,B 0.000,C -6.000}
DECL LDAT LCPDATP210={VEL 0.076,ACC 100,APO_DIST 5,APO_FAC 50.0,ORI_TYP #VAR,CIRC_TYP #BASE,JERK_FAC 50.0}
DECL FDAT FP210={TOOL_NO 2,BASE_NO 8,IPO_FRAME #BASE,POINT2[] " ",TQ_STATE FALSE}
DECL E6POS XP210={X 50.000,Y 145.240,Z -80.570,A 0.000,B 0.000,C -31.000}
DECL LDAT LCPDATP211={VEL 0.076,ACC 100,APO_DIST 5,APO_FAC 50.0,ORI_TYP #VAR,CIRC_TYP #BASE,JERK_FAC 50.0}
DECL FDAT FP211={TOOL_NO 2,BASE_NO 8,IPO_FRAME #BASE,POINT2[] " ",TQ_STATE FALSE}
DECL E6POS XP211={X -0.000,Y 145.240,Z -80.570,A 0.000,B 0.000,C -31.000}
DECL LDAT LCPDATP212={VEL 0.076,ACC 100,APO_DIST 5,APO_FAC 50.0,ORI_TYP #VAR,CIRC_TYP #BASE,JERK_FAC 50.0}
DECL FDAT FP212={TOOL_NO 2,BASE_NO 8,IPO_FRAME #BASE,POINT2[] " ",TQ_STATE FALSE}
DECL E6POS XP212={X -50.000,Y 145.240,Z -80.570,A 0.000,B 0.000,C -31.000}
DECL LDAT LCPDATP213={VEL 0.076,ACC 100,APO_DIST 5,APO_FAC 50.0,ORI_TYP #VAR,CIRC_TYP #BASE,JERK_FAC 50.0}
DECL FDAT FP213={TOOL_NO 2,BASE_NO 8,IPO_FRAME #BASE,POINT2[] " ",TQ_STATE FALSE}
DECL E6POS XP213={X -100.000,Y 145.240,Z -80.570,A 0.000,B 0.000,C -31.000}
DECL LDAT LCPDATP214={VEL 0.126,ACC 100,APO_DIST 5,APO_FAC 50.0,ORI_TYP #VAR,CIRC_TYP #BASE,JERK_FAC 50.0}
DECL FDAT FP214={TOOL_NO 2,BASE_NO 8,IPO_FRAME #BASE,POINT2[] " ",TQ_STATE FALSE}
DECL E6POS XP214={X -100.000,Y 168.140,Z -58.030,A 0.000,B 0.000,C -34.000}
DECL LDAT LCPDATP215={VEL 0.126,ACC 100,APO_DIST 5,APO_FAC 50.0,ORI_TYP #VAR,CIRC_TYP #BASE,JERK_FAC 50.0}
DECL FDAT FP215={TOOL_NO 2,BASE_NO 8,IPO_FRAME #BASE,POINT2[] " ",TQ_STATE FALSE}
DECL E6POS XP215={X -50.000,Y 168.140,Z -58.030,A 0.000,B 0.000,C -34.000}
DECL LDAT LCPDATP216={VEL 0.126,ACC 100,APO_DIST 5,APO_FAC 50.0,ORI_TYP #VAR,CIRC_TYP #BASE,JERK_FAC 50.0}
DECL FDAT FP216={TOOL_NO 2,BASE_NO 8,IPO_FRAME #BASE,POINT2[] " ",TQ_STATE FALSE}
DECL E6POS XP216={X -0.000,Y 168.140,Z -58.030,A 0.000,B 0.000,C -34.000}
DECL LDAT LCPDATP217={VEL 0.126,ACC 100,APO_DIST 5,APO_FAC 50.0,ORI_TYP #VAR,CIRC_TYP #BASE,JERK_FAC 50.0}
DECL FDAT FP217={TOOL_NO 2,BASE_NO 8,IPO_FRAME #BASE,POINT2[] " ",TQ_STATE FALSE}
DECL E6POS XP217={X 50.000,Y 168.140,Z -58.030,A 0.000,B 0.000,C -34.000}
DECL LDAT LCPDATP218={VEL 0.13,ACC 100,APO_DIST 5,APO_FAC 50.0,ORI_TYP #VAR,CIRC_TYP #BASE,JERK_FAC 50.0}
DECL FDAT FP218={TOOL_NO 2,BASE_NO 8,IPO_FRAME #BASE,POINT2[] " ",TQ_STATE FALSE}
DECL E6POS XP218={X 50.000,Y 200.790,Z -31.380,A 0.000,B 0.000,C -32.000}
DECL LDAT LCPDATP219={VEL 0.13,ACC 100,APO_DIST 5,APO_FAC 50.0,ORI_TYP #VAR,CIRC_TYP #BASE,JERK_FAC 50.0}
DECL FDAT FP219={TOOL_NO 2,BASE_NO 8,IPO_FRAME #BASE,POINT2[] " ",TQ_STATE FALSE}
DECL E6POS XP219={X -0.000,Y 200.790,Z -31.380,A 0.000,B 0.000,C -32.000}
DECL LDAT LCPDATP220={VEL 0.13,ACC 100,APO_DIST 5,APO_FAC 50.0,ORI_TYP #VAR,CIRC_TYP #BASE,JERK_FAC 50.0}
DECL FDAT FP220={TOOL_NO 2,BASE_NO 8,IPO_FRAME #BASE,POINT2[] " ",TQ_STATE FALSE}
DECL E6POS XP220={X -50.000,Y 200.790,Z -31.380,A 0.000,B 0.000,C -32.000}
DECL LDAT LCPDATP221={VEL 0.13,ACC 100,APO_DIST 5,APO_FAC 50.0,ORI_TYP #VAR,CIRC_TYP #BASE,JERK_FAC 50.0}
DECL FDAT FP221={TOOL_NO 2,BASE_NO 8,IPO_FRAME #BASE,POINT2[] " ",TQ_STATE FALSE}
DECL E6POS XP221={X -100.000,Y 200.790,Z -31.380,A 0.000,B 0.000,C -32.000}
DECL LDAT LCPDATP222={VEL 0.106,ACC 100,APO_DIST 5,APO_FAC 50.0,ORI_TYP #VAR,CIRC_TYP #BASE,JERK_FAC 50.0}
DECL FDAT FP222={TOOL_NO 2,BASE_NO 8,IPO_FRAME #BASE,POINT2[] " ",TQ_STATE FALSE}
DECL E6POS XP222={X -100.000,Y 225.990,Z -88.130,A 0.000,B 0.000,C -8.000}
DECL LDAT LCPDATP223={VEL 0.106,ACC 100,APO_DIST 5,APO_FAC 50.0,ORI_TYP #VAR,CIRC_TYP #BASE,JERK_FAC 50.0}
DECL FDAT FP223={TOOL_NO 2,BASE_NO 8,IPO_FRAME #BASE,POINT2[] " ",TQ_STATE FALSE}
DECL E6POS XP223={X -50.000,Y 225.990,Z -88.130,A 0.000,B 0.000,C -8.000}
DECL LDAT LCPDATP224={VEL 0.106,ACC 100,APO_DIST 5,APO_FAC 50.0,ORI_TYP #VAR,CIRC_TYP #BASE,JERK_FAC 50.0}
DECL FDAT FP224={TOOL_NO 2,BASE_NO 8,IPO_FRAME #BASE,POINT2[] " ",TQ_STATE FALSE}
DECL E6POS XP224={X -0.000,Y 225.990,Z -88.130,A 0.000,B 0.000,C -8.000}
DECL LDAT LCPDATP225={VEL 0.106,ACC 100,APO_DIST 5,APO_FAC 50.0,ORI_TYP #VAR,CIRC_TYP #BASE,JERK_FAC 50.0}
DECL FDAT FP225={TOOL_NO 2,BASE_NO 8,IPO_FRAME #BASE,POINT2[] " ",TQ_STATE FALSE}
DECL E6POS XP225={X 50.000,Y 225.990,Z -88.130,A 0.000,B 0.000,C -8.000}
DECL LDAT LCPDATP226={VEL 0.145,ACC 100,APO_DIST 5,APO_FAC 50.0,ORI_TYP #VAR,CIRC_TYP #BASE,JERK_FAC 50.0}
DECL FDAT FP226={TOOL_NO 2,BASE_NO 8,IPO_FRAME #BASE,POINT2[] " ",TQ_STATE FALSE}
DECL E6POS XP226={X 50.000,Y 209.360,Z -72.860,A 0.000,B 0.000,C -31.000}
DECL LDAT LCPDATP227={VEL 0.145,ACC 100,APO_DIST 5,APO_FAC 50.0,ORI_TYP #VAR,CIRC_TYP #BASE,JERK_FAC 50.0}
DECL FDAT FP227={TOOL_NO 2,BASE_NO 8,IPO_FRAME #BASE,POINT2[] " ",TQ_STATE FALSE}
DECL E6POS XP227={X -0.000,Y 209.360,Z -72.860,A 0.000,B 0.000,C -31.000}
DECL LDAT LCPDATP228={VEL 0.145,ACC 100,APO_DIST 5,APO_FAC 50.0,ORI_TYP #VAR,CIRC_TYP #BASE,JERK_FAC 50.0}
DECL FDAT FP228={TOOL_NO 2,BASE_NO 8,IPO_FRAME #BASE,POINT2[] " ",TQ_STATE FALSE}
DECL E6POS XP228={X -50.000,Y 209.360,Z -72.860,A 0.000,B 0.000,C -31.000}
DECL LDAT LCPDATP229={VEL 0.145,ACC 100,APO_DIST 5,APO_FAC 50.0,ORI_TYP #VAR,CIRC_TYP #BASE,JERK_FAC 50.0}
DECL FDAT FP229={TOOL_NO 2,BASE_NO 8,IPO_FRAME #BASE,POINT2[] " ",TQ_STATE FALSE}
DECL E6POS XP229={X -100.000,Y 209.360,Z -72.860,A 0.000,B 0.000,C -31.000}
DECL LDAT LCPDATP230={VEL 0.1,ACC 100,APO_DIST 5,APO_FAC 50.0,ORI_TYP #VAR,CIRC_TYP #BASE,JERK_FAC 50.0}
DECL FDAT FP230={TOOL_NO 2,BASE_NO 8,IPO_FRAME #BASE,POINT2[] " ",TQ_STATE FALSE}
DECL E6POS XP230={X -100.000,Y 244.930,Z -87.900,A 0.000,B 0.000,C -15.000}
DECL LDAT LCPDATP231={VEL 0.1,ACC 100,APO_DIST 5,APO_FAC 50.0,ORI_TYP #VAR,CIRC_TYP #BASE,JERK_FAC 50.0}
DECL FDAT FP231={TOOL_NO 2,BASE_NO 8,IPO_FRAME #BASE,POINT2[] " ",TQ_STATE FALSE}
DECL E6POS XP231={X -50.000,Y 244.930,Z -87.900,A 0.000,B 0.000,C -15.000}
DECL LDAT LCPDATP232={VEL 0.1,ACC 100,APO_DIST 5,APO_FAC 50.0,ORI_TYP #VAR,CIRC_TYP #BASE,JERK_FAC 50.0}
DECL FDAT FP232={TOOL_NO 2,BASE_NO 8,IPO_FRAME #BASE,POINT2[] " ",TQ_STATE FALSE}
DECL E6POS XP232={X -0.000,Y 244.930,Z -87.900,A 0.000,B 0.000,C -15.000}
DECL LDAT LCPDATP233={VEL 0.1,ACC 100,APO_DIST 5,APO_FAC 50.0,ORI_TYP #VAR,CIRC_TYP #BASE,JERK_FAC 50.0}
DECL FDAT FP233={TOOL_NO 2,BASE_NO 8,IPO_FRAME #BASE,POINT2[] " ",TQ_STATE FALSE}
DECL E6POS XP233={X 50.000,Y 244.930,Z -87.900,A 0.000,B 0.000,C -15.000}
DECL LDAT LCPDATP234={VEL 0.13,ACC 100,APO_DIST 5,APO_FAC 50.0,ORI_TYP #VAR,CIRC_TYP #BASE,JERK_FAC 50.0}
DECL FDAT FP234={TOOL_NO 2,BASE_NO 8,IPO_FRAME #BASE,POINT2[] " ",TQ_STATE FALSE}
DECL E6POS XP234={X 50.000,Y 261.110,Z -60.510,A 0.000,B 0.000,C -19.000}
DECL LDAT LCPDATP235={VEL 0.13,ACC 100,APO_DIST 5,APO_FAC 50.0,ORI_TYP #VAR,CIRC_TYP #BASE,JERK_FAC 50.0}
DECL FDAT FP235={TOOL_NO 2,BASE_NO 8,IPO_FRAME #BASE,POINT2[] " ",TQ_STATE FALSE}
DECL E6POS XP235={X -0.000,Y 261.110,Z -60.510,A 0.000,B 0.000,C -19.000}
DECL LDAT LCPDATP236={VEL 0.13,ACC 100,APO_DIST 5,APO_FAC 50.0,ORI_TYP #VAR,CIRC_TYP #BASE,JERK_FAC 50.0}
DECL FDAT FP236={TOOL_NO 2,BASE_NO 8,IPO_FRAME #BASE,POINT2[] " ",TQ_STATE FALSE}
DECL E6POS XP236={X -50.000,Y 261.110,Z -60.510,A 0.000,B 0.000,C -19.000}
DECL LDAT LCPDATP237={VEL 0.13,ACC 100,APO_DIST 5,APO_FAC 50.0,ORI_TYP #VAR,CIRC_TYP #BASE,JERK_FAC 50.0}
DECL FDAT FP237={TOOL_NO 2,BASE_NO 8,IPO_FRAME #BASE,POINT2[] " ",TQ_STATE FALSE}
DECL E6POS XP237={X -100.000,Y 261.110,Z -60.510,A 0.000,B 0.000,C -19.000}
DECL LDAT LCPDATP238={VEL 0.091,ACC 100,APO_DIST 5,APO_FAC 50.0,ORI_TYP #VAR,CIRC_TYP #BASE,JERK_FAC 50.0}
DECL FDAT FP238={TOOL_NO 2,BASE_NO 8,IPO_FRAME #BASE,POINT2[] " ",TQ_STATE FALSE}
DECL E6POS XP238={X -100.000,Y 287.330,Z -59.260,A 0.000,B 0.000,C -9.000}
DECL LDAT LCPDATP239={VEL 0.091,ACC 100,APO_DIST 5,APO_FAC 50.0,ORI_TYP #VAR,CIRC_TYP #BASE,JERK_FAC 50.0}
DECL FDAT FP239={TOOL_NO 2,BASE_NO 8,IPO_FRAME #BASE,POINT2[] " ",TQ_STATE FALSE}
DECL E6POS XP239={X -50.000,Y 287.330,Z -59.260,A 0.000,B 0.000,C -9.000}
DECL LDAT LCPDATP240={VEL 0.091,ACC 100,APO_DIST 5,APO_FAC 50.0,ORI_TYP #VAR,CIRC_TYP #BASE,JERK_FAC 50.0}
DECL FDAT FP240={TOOL_NO 2,BASE_NO 8,IPO_FRAME #BASE,POINT2[] " ",TQ_STATE FALSE}
DECL E6POS XP240={X -0.000,Y 287.330,Z -59.260,A 0.000,B 0.000,C -9.000}
DECL LDAT LCPDATP241={VEL 0.091,ACC 100,APO_DIST 5,APO_FAC 50.0,ORI_TYP #VAR,CIRC_TYP #BASE,JERK_FAC 50.0}
DECL FDAT FP241={TOOL_NO 2,BASE_NO 8,IPO_FRAME #BASE,POINT2[] " ",TQ_STATE FALSE}
DECL E6POS XP241={X 50.000,Y 287.330,Z -59.260,A 0.000,B 0.000,C -9.000}
DECL LDAT LCPDATP242={VEL 0.5,ACC 100,APO_DIST 5,APO_FAC 50.0,ORI_TYP #VAR,CIRC_TYP #BASE,JERK_FAC 50.0}
DECL FDAT FP242={TOOL_NO 2,BASE_NO 8,IPO_FRAME #BASE,POINT2[] " ",TQ_STATE FALSE}
DECL E6POS XP242={X 100.000,Y 296.710,Z -50.000,A 0.000,B 0.000,C 0.000}
DECL LDAT LCPDATP243={VEL 1.0,ACC 100,APO_DIST 5,APO_FAC 50.0,ORI_TYP #VAR,CIRC_TYP #BASE,JERK_FAC 50.0}
DECL FDAT FP243={TOOL_NO 2,BASE_NO 8,IPO_FRAME #BASE,POINT2[] " ",TQ_STATE FALSE}
DECL E6POS XP243={X 100.000,Y 340.000,Z -20.000,A 0.000,B 0.000,C 0.000}
DECL LDAT LCPDATP244={VEL 1.0,ACC 100,APO_DIST 5,APO_FAC 50.0,ORI_TYP #VAR,CIRC_TYP #BASE,JERK_FAC 50.0}
DECL FDAT FP244={TOOL_NO 2,BASE_NO 8,IPO_FRAME #BASE,POINT2[] " ",TQ_STATE FALSE}
DECL E6POS XP244={X 100.000,Y 340.000,Z -20.000,A 0.000,B 0.000,C 0.000}
;ENDDAT for Routine_2


; Data for Routine_3
DECL LDAT LCPDATP245={VEL 1.0,ACC 100,APO_DIST 5,APO_FAC 50.0,ORI_TYP #VAR,CIRC_TYP #BASE,JERK_FAC 50.0}
DECL FDAT FP245={TOOL_NO 2,BASE_NO 7,IPO_FRAME #BASE,POINT2[] " ",TQ_STATE FALSE}
DECL E6POS XP245={X 100.000,Y 0.000,Z -100.000,A 0.000,B 0.000,C 0.000}
DECL LDAT LCPDATP246={VEL 0.097,ACC 100,APO_DIST 5,APO_FAC 50.0,ORI_TYP #VAR,CIRC_TYP #BASE,JERK_FAC 50.0}
DECL FDAT FP246={TOOL_NO 2,BASE_NO 7,IPO_FRAME #BASE,POINT2[] " ",TQ_STATE FALSE}
DECL E6POS XP246={X 50.000,Y 7.060,Z -40.840,A 0.000,B 0.000,C -5.000}
DECL LDAT LCPDATP247={VEL 0.097,ACC 100,APO_DIST 5,APO_FAC 50.0,ORI_TYP #VAR,CIRC_TYP #BASE,JERK_FAC 50.0}
DECL FDAT FP247={TOOL_NO 2,BASE_NO 7,IPO_FRAME #BASE,POINT2[] " ",TQ_STATE FALSE}
DECL E6POS XP247={X -0.000,Y 7.060,Z -40.840,A 0.000,B 0.000,C -5.000}
DECL LDAT LCPDATP248={VEL 0.097,ACC 100,APO_DIST 5,APO_FAC 50.0,ORI_TYP #VAR,CIRC_TYP #BASE,JERK_FAC 50.0}
DECL FDAT FP248={TOOL_NO 2,BASE_NO 7,IPO_FRAME #BASE,POINT2[] " ",TQ_STATE FALSE}
DECL E6POS XP248={X -50.000,Y 7.060,Z -40.840,A 0.000,B 0.000,C -5.000}
DECL LDAT LCPDATP249={VEL 0.097,ACC 100,APO_DIST 5,APO_FAC 50.0,ORI_TYP #VAR,CIRC_TYP #BASE,JERK_FAC 50.0}
DECL FDAT FP249={TOOL_NO 2,BASE_NO 7,IPO_FRAME #BASE,POINT2[] " ",TQ_STATE FALSE}
DECL E6POS XP249={X -100.000,Y 7.060,Z -40.840,A 0.000,B 0.000,C -5.000}
DECL LDAT LCPDATP250={VEL 0.144,ACC 100,APO_DIST 5,APO_FAC 50.0,ORI_TYP #VAR,CIRC_TYP #BASE,JERK_FAC 50.0}
DECL FDAT FP250={TOOL_NO 2,BASE_NO 7,IPO_FRAME #BASE,POINT2[] " ",TQ_STATE FALSE}
DECL E6POS XP250={X -100.000,Y 5.010,Z -45.320,A 0.000,B 0.000,C -25.000}
DECL LDAT LCPDATP251={VEL 0.144,ACC 100,APO_DIST 5,APO_FAC 50.0,ORI_TYP #VAR,CIRC_TYP #BASE,JERK_FAC 50.0}
DECL FDAT FP251={TOOL_NO 2,BASE_NO 7,IPO_FRAME #BASE,POINT2[] " ",TQ_STATE FALSE}
DECL E6POS XP251={X -50.000,Y 5.010,Z -45.320,A 0.000,B 0.000,C -25.000}
DECL LDAT LCPDATP252={VEL 0.144,ACC 100,APO_DIST 5,APO_FAC 50.0,ORI_TYP #VAR,CIRC_TYP #BASE,JERK_FAC 50.0}
DECL FDAT FP252={TOOL_NO 2,BASE_NO 7,IPO_FRAME #BASE,POINT2[] " ",TQ_STATE FALSE}
DECL E6POS XP252={X -0.000,Y 5.010,Z -45.320,A 0.000,B 0.000,C -25.000}
DECL LDAT LCPDATP253={VEL 0.144,ACC 100,APO_DIST 5,APO_FAC 50.0,ORI_TYP #VAR,CIRC_TYP #BASE,JERK_FAC 50.0}
DECL FDAT FP253={TOOL_NO 2,BASE_NO 7,IPO_FRAME #BASE,POINT2[] " ",TQ_STATE FALSE}
DECL E6POS XP253={X 50.000,Y 5.010,Z -45.320,A 0.000,B 0.000,C -25.000}
DECL LDAT LCPDATP254={VEL 0.084,ACC 100,APO_DIST 5,APO_FAC 50.0,ORI_TYP #VAR,CIRC_TYP #BASE,JERK_FAC 50.0}
DECL FDAT FP254={TOOL_NO 2,BASE_NO 7,IPO_FRAME #BASE,POINT2[] " ",TQ_STATE FALSE}
DECL E6POS XP254={X 50.000,Y 26.740,Z -40.660,A 0.000,B 0.000,C -19.000}
DECL LDAT LCPDATP255={VEL 0.084,ACC 100,APO_DIST 5,APO_FAC 50.0,ORI_TYP #VAR,CIRC_TYP #BASE,JERK_FAC 50.0}
DECL FDAT FP255={TOOL_NO 2,BASE_NO 7,IPO_FRAME #BASE,POINT2[] " ",TQ_STATE FALSE}
DECL E6POS XP255={X -0.000,Y 26.740,Z -40.660,A 0.000,B 0.000,C -19.000}
DECL LDAT LCPDATP256={VEL 0.084,ACC 100,APO_DIST 5,APO_FAC 50.0,ORI_TYP #VAR,CIRC_TYP #BASE,JERK_FAC 50.0}
DECL FDAT FP256={TOOL_NO 2,BASE_NO 7,IPO_FRAME #BASE,POINT2[] " ",TQ_STATE FALSE}
DECL E6POS XP256={X -50.000,Y 26.740,Z -40.660,A 0.000,B 0.000,C -19.000}
DECL LDAT LCPDATP257={VEL 0.084,ACC 100,APO_DIST 5,APO_FAC 50.0,ORI_TYP #VAR,CIRC_TYP #BASE,JERK_FAC 50.0}
DECL FDAT FP257={TOOL_NO 2,BASE_NO 7,IPO_FRAME #BASE,POINT2[] " ",TQ_STATE FALSE}
DECL E6POS XP257={X -100.000,Y 26.740,Z -40.660,A 0.000,B 0.000,C -19.000}
DECL LDAT LCPDATP258={VEL 0.05,ACC 100,APO_DIST 5,APO_FAC 50.0,ORI_TYP #VAR,CIRC_TYP #BASE,JERK_FAC 50.0}
DECL FDAT FP258={TOOL_NO 2,BASE_NO 7,IPO_FRAME #BASE,POINT2[] " ",TQ_STATE FALSE}
DECL E6POS XP258={X -100.000,Y 19.360,Z -79.990,A 0.000,B 0.000,C -26.000}
DECL LDAT LCPDATP259={VEL 0.05,ACC 100,APO_DIST 5,APO_FAC 50.0,ORI_TYP #VAR,CIRC_TYP #BASE,JERK_FAC 50.0}
DECL FDAT FP259={TOOL_NO 2,BASE_NO 7,IPO_FRAME #BASE,POINT2[] " ",TQ_STATE FALSE}
DECL E6POS XP259={X -50.000,Y 19.360,Z -79.990,A 0.000,B 0.000,C -26.000}
DECL LDAT LCPDATP260={VEL 0.05,ACC 100,APO_DIST 5,APO_FAC 50.0,ORI_TYP #VAR,CIRC_TYP #BASE,JERK_FAC 50.0}
DECL FDAT FP260={TOOL_NO 2,BASE_NO 7,IPO_FRAME #BASE,POINT2[] " ",TQ_STATE FALSE}
DECL E6POS XP260={X -0.000,Y 19.360,Z -79.990,A 0.000,B 0.000,C -26.000}
DECL LDAT LCPDATP261={VEL 0.05,ACC 100,APO_DIST 5,APO_FAC 50.0,ORI_TYP #VAR,CIRC_TYP #BASE,JERK_FAC 50.0}
DECL FDAT FP261={TOOL_NO 2,BASE_NO 7,IPO_FRAME #BASE,POINT2[] " ",TQ_STATE FALSE}
DECL E6POS XP261={X 50.000,Y 19.360,Z -79.990,A 0.000,B 0.000,C -26.000}
DECL LDAT LCPDATP262={VEL 0.077,ACC 100,APO_DIST 5,APO_FAC 50.0,ORI_TYP #VAR,CIRC_TYP #BASE,JERK_FAC 50.0}
DECL FDAT FP262={TOOL_NO 2,BASE_NO 7,IPO_FRAME #BASE,POINT2[] " ",TQ_STATE FALSE}
DECL E6POS XP262={X 50.000,Y 64.350,Z -47.530,A 0.000,B 0.000,C -8.000}
DECL LDAT LCPDATP263={VEL 0.077,ACC 100,APO_DIST 5,APO_FAC 50.0,ORI_TYP #VAR,CIRC_TYP #BASE,JERK_FAC 50.0}
DECL FDAT FP263={TOOL_NO 2,BASE_NO 7,IPO_FRAME #BASE,POINT2[] " ",TQ_STATE FALSE}
DECL E6POS XP263={X -0.000,Y 64.350,Z -47.530,A 0.000,B 0.000,C -8.000}
DECL LDAT LCPDATP264={VEL 0.077,ACC 100,APO_DIST 5,APO_FAC 50.0,ORI_TYP #VAR,CIRC_TYP #BASE,JERK_FAC 50.0}
DECL FDAT FP264={TOOL_NO 2,BASE_NO 7,IPO_FRAME #BASE,POINT2[] " ",TQ_STATE FALSE}
DECL E6POS XP264={X -50.000,Y 64.350,Z -47.530,A 0.000,B 0.000,C -8.000}
DECL LDAT LCPDATP265={VEL 0.077,ACC 100,APO_DIST 5,APO_FAC 50.0,ORI_TYP #VAR,CIRC_TYP #BASE,JERK_FAC 50.0}
DECL FDAT FP265={TOOL_NO 2,BASE_NO 7,IPO_FRAME #BASE,POINT2[] " ",TQ_STATE FALSE}
DECL E6POS XP265={X -100.000,Y 64.350,Z -47.530,A 0.000,B 0.000,C -8.000}
DECL LDAT LCPDATP266={VEL 0.091,ACC 100,APO_DIST 5,APO_FAC 50.0,ORI_TYP #VAR,CIRC_TYP #BASE,JERK_FAC 50.0}
DECL FDAT FP266={TOOL_NO 2,BASE_NO 7,IPO_FRAME #BASE,POINT2[] " ",TQ_STATE FALSE}
DECL E6POS XP266={X -100.000,Y 33.940,Z -75.240,A 0.000,B 0.000,C -36.000}
DECL LDAT LCPDATP267={VEL 0.091,ACC 100,APO_DIST 5,APO_FAC 50.0,ORI_TYP #VAR,CIRC_TYP #BASE,JERK_FAC 50.0}
DECL FDAT FP267={TOOL_NO 2,BASE_NO 7,IPO_FRAME #BASE,POINT2[] " ",TQ_STATE FALSE}
DECL E6POS XP267={X -50.000,Y 33.940,Z -75.240,A 0.000,B 0.000,C -36.000}
DECL LDAT LCPDATP268={VEL 0.091,ACC 100,APO_DIST 5,APO_FAC 50.0,ORI_TYP #VAR,CIRC_TYP #BASE,JERK_FAC 50.0}
DECL FDAT FP268={TOOL_NO 2,BASE_NO 7,IPO_FRAME #BASE,POINT2[] " ",TQ_STATE FALSE}
DECL E6POS XP268={X -0.000,Y 33.940,Z -75.240,A 0.000,B 0.000,C -36.000}
DECL LDAT LCPDATP269={VEL 0.091,ACC 100,APO_DIST 5,APO_FAC 50.0,ORI_TYP #VAR,CIRC_TYP #BASE,JERK_FAC 50.0}
DECL FDAT FP269={TOOL_NO 2,BASE_NO 7,IPO_FRAME #BASE,POINT2[] " ",TQ_STATE FALSE}
DECL E6POS XP269={X 50.000,Y 33.940,Z -75.240,A 0.000,B 0.000,C -36.000}
DECL LDAT LCPDATP270={VEL 0.058,ACC 100,APO_DIST 5,APO_FAC 50.0,ORI_TYP #VAR,CIRC_TYP #BASE,JERK_FAC 50.0}
DECL FDAT FP270={TOOL_NO 2,BASE_NO 7,IPO_FRAME #BASE,POINT2[] " ",TQ_STATE FALSE}
DECL E6POS XP270={X 50.000,Y 90.000,Z -60.860,A 0.000,B 0.000,C -11.000}
DECL LDAT LCPDATP271={VEL 0.058,ACC 100,APO_DIST 5,APO_FAC 50.0,ORI_TYP #VAR,CIRC_TYP #BASE,JERK_FAC 50.0}
DECL FDAT FP271={TOOL_NO 2,BASE_NO 7,IPO_FRAME #BASE,POINT2[] " ",TQ_STATE FALSE}
DECL E6POS XP271={X -0.000,Y 90.000,Z -60.860,A 0.000,B 0.000,C -11.000}
DECL LDAT LCPDATP272={VEL 0.058,ACC 100,APO_DIST 5,APO_FAC 50.0,ORI_TYP #VAR,CIRC_TYP #BASE,JERK_FAC 50.0}
DECL FDAT FP272={TOOL_NO 2,BASE_NO 7,IPO_FRAME #BASE,POINT2[] " ",TQ_STATE FALSE}
DECL E6POS XP272={X -50.000,Y 90.000,Z -60.860,A 0.000,B 0.000,C -11.000}
DECL LDAT LCPDATP273={VEL 0.058,ACC 100,APO_DIST 5,APO_FAC 50.0,ORI_TYP #VAR,CIRC_TYP #BASE,JERK_FAC 50.0}
DECL FDAT FP273={TOOL_NO 2,BASE_NO 7,IPO_FRAME #BASE,POINT2[] " ",TQ_STATE FALSE}
DECL E6POS XP273={X -100.000,Y 90.000,Z -60.860,A 0.000,B 0.000,C -11.000}
DECL LDAT LCPDATP274={VEL 0.08,ACC 100,APO_DIST 5,APO_FAC 50.0,ORI_TYP #VAR,CIRC_TYP #BASE,JERK_FAC 50.0}
DECL FDAT FP274={TOOL_NO 2,BASE_NO 7,IPO_FRAME #BASE,POINT2[] " ",TQ_STATE FALSE}
DECL E6POS XP274={X -100.000,Y 108.240,Z -77.420,A 0.000,B 0.000,C -7.000}
DECL LDAT LCPDATP275={VEL 0.08,ACC 100,APO_DIST 5,APO_FAC 50.0,ORI_TYP #VAR,CIRC_TYP #BASE,JERK_FAC 50.0}
DECL FDAT FP275={TOOL_NO 2,BASE_NO 7,IPO_FRAME #BASE,POINT2[] " ",TQ_STATE FALSE}
DECL E6POS XP275={X -50.000,Y 108.240,Z -77.420,A 0.000,B 0.000,C -7.000}
DECL LDAT LCPDATP276={VEL 0.08,ACC 100,APO_DIST 5,APO_FAC 50.0,ORI_TYP #VAR,CIRC_TYP #BASE,JERK_FAC 50.0}
DECL FDAT FP276={TOOL_NO 2,BASE_NO 7,IPO_FRAME #BASE,POINT2[] " ",TQ_STATE FALSE}
DECL E6POS XP276={X -0.000,Y 108.240,Z -77.420,A 0.000,B 0.000,C -7.000}
DECL LDAT LCPDATP277={VEL 0.08,ACC 100,APO_DIST 5,APO_FAC 50.0,ORI_TYP #VAR,CIRC_TYP #BASE,JERK_FAC 50.0}
DECL FDAT FP277={TOOL_NO 2,BASE_NO 7,IPO_FRAME #BASE,POINT2[] " ",TQ_STATE FALSE}
DECL E6POS XP277={X 50.000,Y 108.240,Z -77.420,A 0.000,B 0.000,C -7.000}
DECL LDAT LCPDATP278={VEL 0.079,ACC 100,APO_DIST 5,APO_FAC 50.0,ORI_TYP #VAR,CIRC_TYP #BASE,JERK_FAC 50.0}
DECL FDAT FP278={TOOL_NO 2,BASE_NO 7,IPO_FRAME #BASE,POINT2[] " ",TQ_STATE FALSE}
DECL E6POS XP278={X 50.000,Y 111.620,Z -37.420,A 0.000,B 0.000,C -27.000}
DECL LDAT LCPDATP279={VEL 0.079,ACC 100,APO_DIST 5,APO_FAC 50.0,ORI_TYP #VAR,CIRC_TYP #BASE,JERK_FAC 50.0}
DECL FDAT FP279={TOOL_NO 2,BASE_NO 7,IPO_FRAME #BASE,POINT2[] " ",TQ_STATE FALSE}
DECL E6POS XP279={X -0.000,Y 111.620,Z -37.420,A 0.000,B 0.000,C -27.000}
DECL LDAT LCPDATP280={VEL 0.079,ACC 100,APO_DIST 5,APO_FAC 50.0,ORI_TYP #VAR,CIRC_TYP #BASE,JERK_FAC 50.0}
DECL FDAT FP280={TOOL_NO 2,BASE_NO 7,IPO_FRAME #BASE,POINT2[] " ",TQ_STATE FALSE}
DECL E6POS XP280={X -50.000,Y 111.620,Z -37.420,A 0.000,B 0.000,C -27.000}
DECL LDAT LCPDATP281={VEL 0.079,ACC 100,APO_DIST 5,APO_FAC 50.0,ORI_TYP #VAR,CIRC_TYP #BASE,JERK_FAC 50.0}
DECL FDAT FP281={TOOL_NO 2,BASE_NO 7,IPO_FRAME #BASE,POINT2[] " ",TQ_STATE FALSE}
DECL E6POS XP281={X -100.000,Y 111.620,Z -37.420,A 0.000,B 0.000,C -27.000}
DECL LDAT LCPDATP282={VEL 0.134,ACC 100,APO_DIST 5,APO_FAC 50.0,ORI_TYP #VAR,CIRC_TYP #BASE,JERK_FAC 50.0}
DECL FDAT FP282={TOOL_NO 2,BASE_NO 7,IPO_FRAME #BASE,POINT2[] " ",TQ_STATE FALSE}
DECL E6POS XP282={X -100.000,Y 124.930,Z -80.750,A 0.000,B 0.000,C -16.000}
DECL LDAT LCPDATP283={VEL 0.134,ACC 100,APO_DIST 5,APO_FAC 50.0,ORI_TYP #VAR,CIRC_TYP #BASE,JERK_FAC 50.0}
DECL FDAT FP283={TOOL_NO 2,BASE_NO 7,IPO_FRAME #BASE,POINT2[] " ",TQ_STATE FALSE}
DECL E6POS XP283={X -50.000,Y 124.930,Z -80.750,A 0.000,B 0.000,C -16.000}
DECL LDAT LCPDATP284={VEL 0.134,ACC 100,APO_DIST 5,APO_FAC 50.0,ORI_TYP #VAR,CIRC_TYP #BASE,JERK_FAC 50.0}
DECL FDAT FP284={TOOL_NO 2,BASE_NO 7,IPO_FRAME #BASE,POINT2[] " ",TQ_STATE FALSE}
DECL E6POS XP284={X -0.000,Y 124.930,Z -80.750,A 0.000,B 0.000,C -16.000}
DECL LDAT LCPDATP285={VEL 0.134,ACC 100,APO_DIST 5,APO_FAC 50.0,ORI_TYP #VAR,CIRC_TYP #BASE,JERK_FAC 50.0}
DECL FDAT FP285={TOOL_NO 2,BASE_NO 7,IPO_FRAME #BASE,POINT2[] " ",TQ_STATE FALSE}
DECL E6POS XP285={X 50.000,Y 124.930,Z -80.750,A 0.000,B 0.000,C -16.000}
DECL LDAT LCPDATP286={VEL 0.141,ACC 100,APO_DIST 5,APO_FAC 50.0,ORI_TYP #VAR,CIRC_TYP #BASE,JERK_FAC 50.0}
DECL FDAT FP286={TOOL_NO 2,BASE_NO 7,IPO_FRAME #BASE,POINT2[] " ",TQ_STATE FALSE}
DECL E6POS XP286={X 50.000,Y 137.040,Z -31.150,A 0.000,B 0.000,C -37.000}
DECL LDAT LCPDATP287={VEL 0.141,ACC 100,APO_DIST 5,APO_FAC 50.0,ORI_TYP #VAR,CIRC_TYP #BASE,JERK_FAC 50.0}
DECL FDAT FP287={TOOL_NO 2,BASE_NO 7,IPO_FRAME #BASE,POINT2[] " ",TQ_STATE FALSE}
DECL E6POS XP287={X -0.000,Y 137.040,Z -31.150,A 0.000,B 0.000,C -37.000}
DECL LDAT LCPDATP288={VEL 0.141,ACC 100,APO_DIST 5,APO_FAC 50.0,ORI_TYP #VAR,CIRC_TYP #BASE,JERK_FAC 50.0}
DECL FDAT FP288={TOOL_NO 2,BASE_NO 7,IPO_FRAME #BASE,POINT2[] " ",TQ_STATE FALSE}
DECL E6POS XP288={X -50.000,Y 137.040,Z -31.150,A 0.000,B 0.000,C -37.000}
DECL LDAT LCPDATP289={VEL 0.141,ACC 100,APO_DIST 5,APO_FAC 50.0,ORI_TYP #VAR,CIRC_TYP #BASE,JERK_FAC 50.0}
DECL FDAT FP289={TOOL_NO 2,BASE_NO 7,IPO_FRAME #BASE,POINT2[] " ",TQ_STATE FALSE}
DECL E6POS XP289={X -100.000,Y 137.040,Z -31.150,A 0.000,B 0.000,C -37.000}
DECL LDAT LCPDATP290={VEL 0.058,ACC 100,APO_DIST 5,APO_FAC 50.0,ORI_TYP #VAR,CIRC_TYP #BASE,JERK_FAC 50.0}
DECL FDAT FP290={TOOL_NO 2,BASE_NO 7,IPO_FRAME #BASE,POINT2[] " ",TQ_STATE FALSE}
DECL E6POS XP290={X -100.000,Y 144.670,Z -47.260,A 0.000,B 0.000,C -34.000}
DECL LDAT LCPDATP291={VEL 0.058,ACC 100,APO_DIST 5,APO_FAC 50.0,ORI_TYP #VAR,CIRC_TYP #BASE,JERK_FAC 50.0}
DECL FDAT FP291={TOOL_NO 2,BASE_NO 7,IPO_FRAME #BASE,POINT2[] " ",TQ_STATE FALSE}
DECL E6POS XP291={X -50.000,Y 144.670,Z -47.260,A 0.000,B 0.000,C -34.000}
DECL LDAT LCPDATP292={VEL 0.058,ACC 100,APO_DIST 5,APO_FAC 50.0,ORI_TYP #VAR,CIRC_TYP #BASE,JERK_FAC 50.0}
DECL FDAT FP292={TOOL_NO 2,BASE_NO 7,IPO_FRAME #BASE,POINT2[] " ",TQ_STATE FALSE}
DECL E6POS XP292={X -0.000,Y 144.670,Z -47.260,A 0.000,B 0.000,C -34.000}
DECL LDAT LCPDATP293={VEL 0.058,ACC 100,APO_DIST 5,APO_FAC 50.0,ORI_TYP #VAR,CIRC_TYP #BASE,JERK_FAC 50.0}
DECL FDAT FP293={TOOL_NO 2,BASE_NO 7,IPO_FRAME #BASE,POINT2[] " ",TQ_STATE FALSE}
DECL E6POS XP293={X 50.000,Y 144.670,Z -47.260,A 0.000,B 0.000,C -34.000}
DECL LDAT LCPDATP294={VEL 0.127,ACC 100,APO_DIST 5,APO_FAC 50.0,ORI_TYP #VAR,CIRC_TYP #BASE,JERK_FAC 50.0}
DECL FDAT FP294={TOOL_NO 2,BASE_NO 7,IPO_FRAME #BASE,POINT2[] " ",TQ_STATE FALSE}
DECL E6POS XP294={X 50.000,Y 175.030,Z -41.080,A 0.000,B 0.000,C -21.000}
DECL LDAT LCPDATP295={VEL 0.127,ACC 100,APO_DIST 5,APO_FAC 50.0,ORI_TYP #VAR,CIRC_TYP #BASE,JERK_FAC 50.0}
DECL FDAT FP295={TOOL_NO 2,BASE_NO 7,IPO_FRAME #BASE,POINT2[] " ",TQ_STATE FALSE}
DECL E6POS XP295={X -0.000,Y 175.030,Z -41.080,A 0.000,B 0.000,C -21.000}
DECL LDAT LCPDATP296={VEL 0.127,ACC 100,APO_DIST 5,APO_FAC 50.0,ORI_TYP #VAR,CIRC_TYP #BASE,JERK_FAC 50.0}
DECL FDAT FP296={TOOL_NO 2,BASE_NO 7,IPO_FRAME #BASE,POINT2[] " ",TQ_STATE FALSE}
DECL E6POS XP296={X -50.000,Y 175.030,Z -41.080,A 0.000,B 0.000,C -21.000}
DECL LDAT LCPDATP297={VEL 0.127,ACC 100,APO_DIST 5,APO_FAC 50.0,ORI_TYP #VAR,CIRC_TYP #BASE,JERK_FAC 50.0}
DECL FDAT FP297={TOOL_NO 2,BASE_NO 7,IPO_FRAME #BASE,POINT2[] " ",TQ_STATE FALSE}
DECL E6POS XP297={X -100.000,Y 175.030,Z -41.080,A 0.000,B 0.000,C -21.000}
DECL LDAT LCPDATP298={VEL 0.052,ACC 100,APO_DIST 5,APO_FAC 50.0,ORI_TYP #VAR,CIRC_TYP #BASE,JERK_FAC 50.0}
DECL FDAT FP298={TOOL_NO 2,BASE_NO 7,IPO_FRAME #BASE,POINT2[] " ",TQ_STATE FALSE}
DECL E6POS XP298={X -100.000,Y 200.830,Z -37.720,A 0.000,B 0.000,C -7.000}
DECL LDAT LCPDATP299={VEL 0.052,ACC 100,APO_DIST 5,APO_FAC 50.0,ORI_TYP #VAR,CIRC_TYP #BASE,JERK_FAC 50.0}
DECL FDAT FP299={TOOL_NO 2,BASE_NO 7,IPO_FRAME #BASE,POINT2[] " ",TQ_STATE FALSE}
DECL E6POS XP299={X -50.000,Y 200.830,Z -37.720,A 0.000,B 0.000,C -7.000}
DECL LDAT LCPDATP300={VEL 0.052,ACC 100,APO_DIST 5,APO_FAC 50.0,ORI_TYP #VAR,CIRC_TYP #BASE,JERK_FAC 50.0}
DECL FDAT FP300={TOOL_NO 2,BASE_NO 7,IPO_FRAME #BASE,POINT2[] " ",TQ_STATE FALSE}
DECL E6POS XP300={X -0.000,Y 200.830,Z -37.720,A 0.000,B 0.000,C -7.000}
DECL LDAT LCPDATP301={VEL 0.052,ACC 100,APO_DIST 5,APO_FAC 50.0,ORI_TYP #VAR,CIRC_TYP #BASE,JERK_FAC 50.0}
DECL FDAT FP301={TOOL_NO 2,BASE_NO 7,IPO_FRAME #BASE,POINT2[] " ",TQ_STATE FALSE}
DECL E6POS XP301={X 50.000,Y 200.830,Z -37.720,A 0.000,B 0.000,C -7.000}
DECL LDAT LCPDATP302={VEL 0.067,ACC 100,APO_DIST 5,APO_FAC 50.0,ORI_TYP #VAR,CIRC_TYP #BASE,JERK_FAC 50.0}
DECL FDAT FP302={TOOL_NO 2,BASE_NO 7,IPO_FRAME #BASE,POINT2[] " ",TQ_STATE FALSE}
DECL E6POS XP302={X 50.000,Y 192.090,Z -58.810,A 0.000,B 0.000,C -27.000}
DECL LDAT LCPDATP303={VEL 0.067,ACC 100,APO_DIST 5,APO_FAC 50.0,ORI_TYP #VAR,CIRC_TYP #BASE,JERK_FAC 50.0}
DECL FDAT FP303={TOOL_NO 2,BASE_NO 7,IPO_FRAME #BASE,POINT2[] " ",TQ_STATE FALSE}
DECL E6POS XP303={X -0.000,Y 192.090,Z -58.810,A 0.000,B 0.000,C -27.000}
DECL LDAT LCPDATP304={VEL 0.067,ACC 100,APO_DIST 5,APO_FAC 50.0,ORI_TYP #VAR,CIRC_TYP #BASE,JERK_FAC 50.0}
DECL FDAT FP304={TOOL_NO 2,BASE_NO 7,IPO_FRAME #BASE,POINT2[] " ",TQ_STATE FALSE}
DECL E6POS XP304={X -50.000,Y 192.090,Z -58.810,A 0.000,B 0.000,C -27.000}
DECL LDAT LCPDATP305={VEL 0.067,ACC 100,APO_DIST 5,APO_FAC 50.0,ORI_TYP #VAR,CIRC_TYP #BASE,JERK_FAC 50.0}
DECL FDAT FP305={TOOL_NO 2,BASE_NO 7,IPO_FRAME #BASE,POINT2[] " ",TQ_STATE FALSE}
DECL E6POS XP305={X -100.000,Y 192.090,Z -58.810,A 0.000,B 0.000,C -27.000}
DECL LDAT LCPDATP306={VEL 0.117,ACC 100,APO_DIST 5,APO_FAC 50.0,ORI_TYP #VAR,CIRC_TYP #BASE,JERK_FAC 50.0}
DECL FDAT FP306={TOOL_NO 2,BASE_NO 7,IPO_FRAME #BASE,POINT2[] " ",TQ_STATE FALSE}
DECL E6POS XP306={X -100.000,Y 235.350,Z -51.990,A 0.000,B 0.000,C -1.000}
DECL LDAT LCPDATP307={VEL 0.117,ACC 100,APO_DIST 5,APO_FAC 50.0,ORI_TYP #VAR,CIRC_TYP #BASE,JERK_FAC 50.0}
DECL FDAT FP307={TOOL_NO 2,BASE_NO 7,IPO_FRAME #BASE,POINT2[] " ",TQ_STATE FALSE}
DECL E6POS XP307={X -50.000,Y 235.350,Z -51.990,A 0.000,B 0.000,C -1.000}
DECL LDAT LCPDATP308={VEL 0.117,ACC 100,APO_DIST 5,APO_FAC 50.0,ORI_TYP #VAR,CIRC_TYP #BASE,JERK_FAC 50.0}
DECL FDAT FP308={TOOL_NO 2,BASE_NO 7,IPO_FRAME #BASE,POINT2[] " ",TQ_STATE FALSE}
DECL E6POS XP308={X -0.000,Y 235.350,Z -51.990,A 0.000,B 0.000,C -1.000}
DECL LDAT LCPDATP309={VEL 0.117,ACC 100,APO_DIST 5,APO_FAC 50.0,ORI_TYP #VAR,CIRC_TYP #BASE,JERK_FAC 50.0}
DECL FDAT FP309={TOOL_NO 2,BASE_NO 7,IPO_FRAME #BASE,POINT2[] " ",TQ_STATE FALSE}
DECL E6POS XP309={X 50.000,Y 235.350,Z -51.990,A 0.000,B 0.000,C -1.000}
DECL LDAT LCPDATP310={VEL 0.138,ACC 100,APO_DIST 5,APO_FAC 50.0,ORI_TYP #VAR,CIRC_TYP #BASE,JERK_FAC 50.0}
DECL FDAT FP310={TOOL_NO 2,BASE_NO 7,IPO_FRAME #BASE,POINT2[] " ",TQ_STATE FALSE}
DECL E6POS XP310={X 50.000,Y 230.810,Z -54.150,A 0.000,B 0.000,C -21.000}
DECL LDAT LCPDATP311={VEL 0.138,ACC 100,APO_DIST 5,APO_FAC 50.0,ORI_TYP #VAR,CIRC_TYP #BASE,JERK_FAC 50.0}
DECL FDAT FP311={TOOL_NO 2,BASE_NO 7,IPO_FRAME #BASE,POINT2[] " ",TQ_STATE FALSE}
DECL E6POS XP311={X -0.000,Y 230.810,Z -54.150,A 0.000,B 0.000,C -21.000}
DECL LDAT LCPDATP312={VEL 0.138,ACC 100,APO_DIST 5,APO_FAC 50.0,ORI_TYP #VAR,CIRC_TYP #BASE,JERK_FAC 50.0}
DECL FDAT FP312={TOOL_NO 2,BASE_NO 7,IPO_FRAME #BASE,POINT2[] " ",TQ_STATE FALSE}
DECL E6POS XP312={X -50.000,Y 230.810,Z -54.150,A 0.000,B 0.000,C -21.000}
DECL LDAT LCPDATP313={VEL 0.138,ACC 100,APO_DIST 5,APO_FAC 50.0,ORI_TYP #VAR,CIRC_TYP #BASE,JERK_FAC 50.0}
DECL FDAT FP313={TOOL_NO 2,BASE_NO 7,IPO_FRAME #BASE,POINT2[] " ",TQ_STATE FALSE}
DECL E6POS XP313={X -100.000,Y 230.810,Z -54.150,A 0.000,B 0.000,C -21.000}
DECL LDAT LCPDATP314={VEL 0.119,ACC 100,APO_DIST 5,APO_FAC 50.0,ORI_TYP #VAR,CIRC_TYP #BASE,JERK_FAC 50.0}
DECL FDAT FP314={TOOL_NO 2,BASE_NO 7,IPO_FRAME #BASE,POINT2[] " ",TQ_STATE FALSE}
DECL E6POS XP314={X -100.000,Y 263.610,Z -66.910,A 0.000,B 0.000,C -3.000}
DECL LDAT LCPDATP315={VEL 0.119,ACC 100,APO_DIST 5,APO_FAC 50.0,ORI_TYP #VAR,CIRC_TYP #BASE,JERK_FAC 50.0}
DECL FDAT FP315={TOOL_NO 2,BASE_NO 7,IPO_FRAME #BASE,POINT2[] " ",TQ_STATE FALSE}
DECL E6POS XP315={X -50.000,Y 263.610,Z -66.910,A 0.000,B 0.000,C -3.000}
DECL LDAT LCPDATP316={VEL 0.119,ACC 100,APO_DIST 5,APO_FAC 50.0,ORI_TYP #VAR,CIRC_TYP #BASE,JERK_FAC 50.0}
DECL FDAT FP316={TOOL_NO 2,BASE_NO 7,IPO_FRAME #BASE,POINT2[] " ",TQ_STATE FALSE}
DECL E6POS XP316={X -0.000,Y 263.610,Z -66.910,A 0.000,B 0.000,C -3.000}
DECL LDAT LCPDATP317={VEL 0.119,ACC 100,APO_DIST 5,APO_FAC 50.0,ORI_TYP #VAR,CIRC_TYP #BASE,JERK_FAC 50.0}
DECL FDAT FP317={TOOL_NO 2,BASE_NO 7,IPO_FRAME #BASE,POINT2[] " ",TQ_STATE FALSE}
DECL E6POS XP317={X 50.000,Y 263.610,Z -66.910,A 0.000,B 0.000,C -3.000}
DECL LDAT LCPDATP318={VEL 0.121,ACC 100,APO_DIST 5,APO_FAC 50.0,ORI_TYP #VAR,CIRC_TYP #BASE,JERK_FAC 50.0}
DECL FDAT FP318={TOOL_NO 2,BASE_NO 7,IPO_FRAME #BASE,POINT2[] " ",TQ_STATE FALSE}
DECL E6POS XP318={X 50.000,Y 261.460,Z -32.910,A 0.000,B 0.000,C -30.000}
DECL LDAT LCPDATP319={VEL 0.121,ACC 100,APO_DIST 5,APO_FAC 50.0,ORI_TYP #VAR,CIRC_TYP #BASE,JERK_FAC 50.0}
DECL FDAT FP319={TOOL_NO 2,BASE_NO 7,IPO_FRAME #BASE,POINT2[] " ",TQ_STATE FALSE}
DECL E6POS XP319={X -0.000,Y 261.460,Z -32.910,A 0.000,B 0.000,C -30.000}
DECL LDAT LCPDATP320={VEL 0.121,ACC 100,APO_DIST 5,APO_FAC 50.0,ORI_TYP #VAR,CIRC_TYP #BASE,JERK_FAC 50.0}
DECL FDAT FP320={TOOL_NO 2,BASE_NO 7,IPO_FRAME #BASE,POINT2[] " ",TQ_STATE FALSE}
DECL E6POS XP320={X -50.000,Y 261.460,Z -32.910,A 0.000,B 0.000,C -30.000}
DECL LDAT LCPDATP321={VEL 0.121,ACC 100,APO_DIST 5,APO_FAC 50.0,ORI_TYP #VAR,CIRC_TYP #BASE,JERK_FAC 50.0}
DECL FDAT FP321={TOOL_NO 2,BASE_NO 7,IPO_FRAME #BASE,POINT2[] " ",TQ_STATE FALSE}
DECL E6POS XP321={X -100.000,Y 261.460,Z -32.910,A 0.000,B 0.000,C -30.000}
DECL LDAT LCPDATP322={VEL 0.059,ACC 100,APO_DIST 5,APO_FAC 50.0,ORI_TYP #VAR,CIRC_TYP #BASE,JERK_FAC 50.0}
DECL FDAT FP322={TOOL_NO 2,BASE_NO 7,IPO_FRAME #BASE,POINT2[] " ",TQ_STATE FALSE}
DECL E6POS XP322={X -100.000,Y 274.650,Z -70.380,A 0.000,B 0.000,C -18.000}
DECL LDAT LCPDATP323={VEL 0.059,ACC 100,APO_DIST 5,APO_FAC 50.0,ORI_TYP #VAR,CIRC_TYP #BASE,JERK_FAC 50.0}
DECL FDAT FP323={TOOL_NO 2,BASE_NO 7,IPO_FRAME #BASE,POINT2[] " ",TQ_STATE FALSE}
DECL E6POS XP323={X -50.000,Y 274.650,Z -70.380,A 0.000,B 0.000,C -18.000}
DECL LDAT LCPDATP324={VEL 0.059,ACC 100,APO_DIST 5,APO_FAC 50.0,ORI_TYP #VAR,CIRC_TYP #BASE,JERK_FAC 50.0}
DECL FDAT FP324={TOOL_NO 2,BASE_NO 7,IPO_FRAME #BASE,POINT2[] " ",TQ_STATE FALSE}
DECL E6POS XP324={X -0.000,Y 274.650,Z -70.380,A 0.000,B 0.000,C -18.000}
DECL LDAT LCPDATP325={VEL 0.059,ACC 100,APO_DIST 5,APO_FAC 50.0,ORI_TYP #VAR,CIRC_TYP #BASE,JERK_FAC 50.0}
DECL FDAT FP325={TOOL_NO 2,BASE_NO 7,IPO_FRAME #BASE,POINT2[] " ",TQ_STATE FALSE}
DECL E6POS XP325={X 50.000,Y 274.650,Z -70.380,A 0.000,B 0.000,C -18.000}
DECL LDAT LCPDATP326={VEL 0.08,ACC 100,APO_DIST 5,APO_FAC 50.0,ORI_TYP #VAR,CIRC_TYP #BASE,JERK_FAC 50.0}
DECL FDAT FP326={TOOL_NO 2,BASE_NO 7,IPO_FRAME #BASE,POINT2[] " ",TQ_STATE FALSE}
DECL E6POS XP326={X 50.000,Y 276.590,Z -87.450,A 0.000,B 0.000,C -23.000}
DECL LDAT LCPDATP327={VEL 0.08,ACC 100,APO_DIST 5,APO_FAC 50.0,ORI_TYP #VAR,CIRC_TYP #BASE,JERK_FAC 50.0}
DECL FDAT FP327={TOOL_NO 2,BASE_NO 7,IPO_FRAME #BASE,POINT2[] " ",TQ_STATE FALSE}
DECL E6POS XP327={X -0.000,Y 276.590,Z -87.450,A 0.000,B 0.000,C -23.000}
DECL LDAT LCPDATP328={VEL 0.08,ACC 100,APO_DIST 5,APO_FAC 50.0,ORI_TYP #VAR,CIRC_TYP #BASE,JERK_FAC 50.0}
DECL FDAT FP328={TOOL_NO 2,BASE_NO 7,IPO_FRAME #BASE,POINT2[] " ",TQ_STATE FALSE}
DECL E6POS XP328={X -50.000,Y 276.590,Z -87.450,A 0.000,B 0.000,C -23.000}
DECL LDAT LCPDATP329={VEL 0.08,ACC 100,APO_DIST 5,APO_FAC 50.0,ORI_TYP #VAR,CIRC_TYP #BASE,JERK_FAC 50.0}
DECL FDAT FP329={TOOL_NO 2,BASE_NO 7,IPO_FRAME #BASE,POINT2[] " ",TQ_STATE FALSE}
DECL E6POS XP329={X -100.000,Y 276.590,Z -87.450,A 0.000,B 0.000,C -23.000}
DECL LDAT LCPDATP330={VEL 0.136,ACC 100,APO_DIST 5,APO_FAC 50.0,ORI_TYP #VAR,CIRC_TYP #BASE,JERK_FAC 50.0}
DECL FDAT FP330={TOOL_NO 2,BASE_NO 7,IPO_FRAME #BASE,POINT2[] " ",TQ_STATE FALSE}
DECL E6POS XP330={X -100.000,Y 311.260,Z -88.350,A 0.000,B 0.000,C -11.000}
DECL LDAT LCPDATP331={VEL 0.136,ACC 100,APO_DIST 5,APO_FAC 50.0,ORI_TYP #VAR,CIRC_TYP #BASE,JERK_FAC 50.0}
DECL FDAT FP331={TOOL_NO 2,BASE_NO 7,IPO_FRAME #BASE,POINT2[] " ",TQ_STATE FALSE}
DECL E6POS XP331={X -50.000,Y 311.260,Z -88.350,A 0.000,B 0.000,C -11.000}
DECL LDAT LCPDATP332={VEL 0.136,ACC 100,APO_DIST 5,APO_FAC 50.0,ORI_TYP #VAR,CIRC_TYP #BASE,JERK_FAC 50.0}
DECL FDAT FP332={TOOL_NO 2,BASE_NO 7,IPO_FRAME #BASE,POINT2[] " ",TQ_STATE FALSE}
DECL E6POS XP332={X -0.000,Y 311.260,Z -88.350,A 0.000,B 0.000,C -11.000}
DECL LDAT LCPDATP333={VEL 0.136,ACC 100,APO_DIST 5,APO_FAC 50.0,ORI_TYP #VAR,CIRC_TYP #BASE,JERK_FAC 50.0}
DECL FDAT FP333={TOOL_NO 2,BASE_NO 7,IPO_FRAME #BASE,POINT2[] " ",TQ_STATE FALSE}
DECL E6POS XP333={X 50.000,Y 311.260,Z -88.350,A 0.000,B 0.000,C -11.000}
DECL LDAT LCPDATP334={VEL 0.5,ACC 100,APO_DIST 5,APO_FAC 50.0,ORI_TYP #VAR,CIRC_TYP #BASE,JERK_FAC 50.0}
DECL FDAT FP334={TOOL_NO 2,BASE_NO 7,IPO_FRAME #BASE,POINT2[] " ",TQ_STATE FALSE}
DECL E6POS XP334={X 100.000,Y 328.430,Z -50.000,A 0.000,B 0.000,C 0.000}
DECL LDAT LCPDATP335={VEL 1.0,ACC 100,APO_DIST 5,APO_FAC 50.0,ORI_TYP #VAR,CIRC_TYP #BASE,JERK_FAC 50.0}
DECL FDAT FP335={TOOL_NO 2,BASE_NO 7,IPO_FRAME #BASE,POINT2[] " ",TQ_STATE FALSE}
DECL E6POS XP335={X 100.000,Y 370.000,Z -20.000,A 0.000,B 0.000,C 0.000}
DECL LDAT LCPDATP336={VEL 1.0,ACC 100,APO_DIST 5,APO_FAC 50.0,ORI_TYP #VAR,CIRC_TYP #BASE,JERK_FAC 50.0}
DECL FDAT FP336={TOOL_NO 2,BASE_NO 7,IPO_FRAME #BASE,POINT2[] " ",TQ_STATE FALSE}
DECL E6POS XP336={X 100.000,Y 370.000,Z -20.000,A 0.000,B 0.000,C 0.000}
;ENDDAT for Routine_3

ENDDAT
